	// SSR
	SSR.SubsystemName	:= mpSSQ^.Position;
	SSR.eReturnCode	:= E_ErrorConv.SubsystemNUMBER_UNKNOWN;

	// Reject telegram	
	M_SendData(
		meChannel := meChannelSrc,
		mMsgType  := E_ITC_MsgTypeConv.SUBSYSTEM_STATUS_REPORT,
		mpData    := ADR(SSR),
		mLen	  := SIZEOF(SSR));
		
	// Unknown SubSystem number received
	DebugMsg := CONCAT('SSQ, unknown SubSystem name received: ', mpSSQ^.Position);
	fbDebugMsg.M_SendErrorMsg(mMessage := DebugMsg);
END_IF
END_METHOD

METHOD PROTECTED M_ProcessTDQ : BOOL
(**************************************************************************************
 *  Application     :   BoxControl Framework
 *  Revision date   :   $Date: 2021-04-08 12:45:11 +0200 (tor, 08 apr 2021) $
 *  Author          :   CDC
 * ------------------------------------------------------------------------------------
 *  © Swisslog AG
 *  Swisslog is not liable for any usage of this source code that is not agreed 
 *  on between Swisslog and the other party. The mandatory legal liability remains 
 *  unaffected.
 * ------------------------------------------------------------------------------------
 *  Revision History: 
 *
 *  VERSION DATE         INITIALS     DESCRIPTION
 *  0.0     DD.MM.YYYY   (name)       (explain customized modifications)
 *
 **************************************************************************************)
VAR_INPUT
	meChannelSrc			: E_MFCS_Channel; // Source communicaton channel
	mpTDQ					: POINTER TO ST_ITC_TDQ; // Pointer to TDQ
	mLen					: UDINT; // Data length
END_VAR

VAR
	mPosition				: ST_PositionIdent ; // Position
	mReturnCode				: E_ErrorConv; // Return code
	mTU_ID_Present			: BOOL; // TU-ID present
	mTU_DataIndex			: DINT; // TU-data index
	mAssignmentID_Present	: BOOL; // Assignment-ID present
	mAssignmentID_Index		: DINT; // Assignment-ID index
END_VAR
// Init
mReturnCode := E_ErrorConv.NO_ERROR_CODE;
M_ProcessTDQ := TRUE;
mTU_ID_Present := FALSE;
mTU_DataIndex := 0;
mAssignmentID_Present := FALSE;
mAssignmentID_Index := 0;

// Get position from telegram
mPosition := F_SearchFunctionPosition( Position := mpTDQ^.Position);

// Order to delete all TU-data
IF mpTDQ^.Code = 1 THEN
	// Check no function number and unknown TU-ID
	IF mpTDQ^.TU_ID = Conveyor.TU_ID_UNKNOWN AND mPosition.eFunctionNumber = 0 THEN
		// Check all TU-Data for DataSets
		FOR mTU_DataIndex := 1 TO Conveyor.NUMBER_OF_TU_DATA BY 1 DO
			// Check if TU-DataSet is used
			IF TU_DataTable[mTU_DataIndex].DataSet.DataPresent THEN	
				// debug message: '11-001-0095-01-1,  TU_DataIndex deleted,  telegram = TDQ,  TU_DataIndex = 5,  TuID = 000012345,  AssignmentID = 999999999'
				DebugMsg := '';
				DebugMsg := CONCAT(DebugMsg, F_AddDividerToSisString(mpTDQ^.Position));
				DebugMsg := CONCAT(DebugMsg, ',  TU_DataIndex deleted');
				DebugMsg := CONCAT(DebugMsg, DebugTextBlocks.TELEGRAM);
				DebugMsg := CONCAT(DebugMsg, 'TDQ');
				DebugMsg := CONCAT(DebugMsg, F_CreateTU_DataString(TU_DataIndex:= mTU_DataIndex));
				fbDebugMsg.M_SendInfoMsg(DebugMsg);
				// Delete TU-Data
				F_DeleteTU_Data(
					TU_DataIndex 	:= mTU_DataIndex, // TU_DataIndex from zone
					NoTTC 			:= FALSE); // No TTC will be sent
			END_IF
		END_FOR

		TDR.Position := mpTDQ^.Position;
		TDR.TU_ID := mpTDQ^.TU_ID;
		TDR.AssignmentID := mpTDQ^.AssignmentID;
		TDR.MsgSequence := mpTDQ^.MsgSequence;
		TDR.ReturnCode := mReturnCode;
		
		M_SendData(
			meChannel := meChannelSrc, 
			mMsgType  := E_ITC_MsgTypeConv.TASK_DELETE_REPORT, 
			mpData    := ADR(TDR),
			mLen	  := SIZEOF(TDR));
		RETURN;
	ELSE
		// Error: Wrong value
		mReturnCode := E_ErrorConv.WRONG_VALUE;
	END_IF
	
// Specific request for TU-ID or position
ELSE
	// Check if an Assignment-ID is present
	mAssignmentID_Present := mpTDQ^.AssignmentID > 0 AND mpTDQ^.AssignmentID < Conveyor.ASSIGNMENT_ID_UNKNOWN;
	
	// Check if a TU-ID is present
	mTU_ID_Present := mpTDQ^.TU_ID <> F_StuffString('', Conveyor.TU_ID_STRINGLENGTH,'0', FALSE) AND
				      mpTDQ^.TU_ID <> F_StuffString('', Conveyor.TU_ID_STRINGLENGTH,' ', FALSE);
	
	// If a valid position is found
	IF mPosition.eFunctionNumber > E_FunctionNumber.F_BEGIN_FUNCTION AND
	   mPosition.ZoneNumber > 0 THEN
		// Get TU-data from zone
		mTU_DataIndex := F_GetTU_DataIndex(
								eFunctionNumber := mPosition.eFunctionNumber, // PositionNumber
								ZoneNumber := mPosition.ZoneNumber); // ZoneNumber
		// A TU index was found
		IF mTU_DataIndex > 0 THEN
			IF mAssignmentID_Present THEN
				// Compare received Assignment ID with the Assignment ID from the position
				IF TU_DataTable[mTU_DataIndex].AssignmentID <> mpTDQ^.AssignmentID THEN
					// Error: Wrong Assignement-ID
					mReturnCode := E_ErrorConv.ASSIGNMENT_ID_WRONG;
				END_IF
			ELSIF mTU_ID_Present THEN
				// Compare received TU ID with the TU ID from the position
				IF TU_DataTable[mTU_DataIndex].TU_ID.ASCII <> mpTDQ^.TU_ID THEN
					// Error: Wrong TU-ID
					mReturnCode := E_ErrorConv.TU_ID_WRONG;
				END_IF
			ELSE
				// Error: Wrong value
				mReturnCode := E_ErrorConv.ID_WRONG;
			END_IF
		ELSE
			// Error: No TU data set available on position
			mReturnCode := E_ErrorConv.EMPTY_TU_DATA_SET;
		END_IF
		
	// Request to subsystem
	ELSIF mpTDQ^.Position <> F_ReduceToAlphaNumeric(SubsystemRegistry.SubsystemName) THEN
		// Error: Position wrong 
		mReturnCode := E_ErrorConv.FUNCTIONNUMBER_UNKNOWN;
		
	// Telegram without function number
	ELSE
		IF mAssignmentID_Present THEN
			// Search TU-data index based on the Assignement-ID in the TU-data table
			mAssignmentID_Index := F_SearchAssignmentId(mpTDQ^.AssignmentID);
		END_IF
		
		IF mTU_ID_Present THEN
			// Search TU-data index based on the TU-ID in the TU-data table
			mTU_DataIndex := F_SearchTU_ByHashCode(mpTDQ^.TU_ID);
		END_IF			
		
		// If an Assignement-ID index is found
		IF mAssignmentID_Index <> 0 THEN
			// Search position belonging to the Assignement-ID index
			// to report last position
			mPosition := F_SearchPositionOfTU_Index(
								TU_DataIndex := mAssignmentID_Index, // TU_DataIndex from zone
								eStartFunctionNumber := E_FunctionNumber.F_BEGIN_FUNCTION + 1); // Start Zone
		// If a TU-data index is found
		ELSIF mTU_DataIndex <> 0 THEN
			// Search position belonging to the TU-data index
			// to report last position
			mPosition := F_SearchPositionOfTU_Index(
								TU_DataIndex := mTU_DataIndex, // TU_DataIndex from zone
								eStartFunctionNumber := E_FunctionNumber.F_BEGIN_FUNCTION + 1); // Start Zone
		ELSE
			IF mAssignmentID_Present THEN
				// Error: Wrong Assignement-ID
				mReturnCode := E_ErrorConv.ASSIGNMENT_ID_WRONG;
			ELSIF mTU_ID_Present THEN
				// Error: Wrong TU-ID
				mReturnCode := E_ErrorConv.TU_ID_WRONG;
			ELSE
				// Error: No data
				mReturnCode := E_ErrorConv.ID_WRONG;
			END_IF
		END_IF
	END_IF
END_IF

// Send task delete report
IF mPosition.eFunctionNumber <> E_FunctionNumber.F_BEGIN_FUNCTION THEN
	TDR.Position := F_ReduceToAlphaNumeric(FunctionRegistry[mPosition.eFunctionNumber].Zone[mPosition.ZoneNumber].ZoneName);
ELSE
	TDR.Position := mpTDQ^.Position;
END_IF
TDR.TU_ID := mpTDQ^.TU_ID;
TDR.AssignmentID := mpTDQ^.AssignmentID;
TDR.MsgSequence := mpTDQ^.MsgSequence;
TDR.ReturnCode := mReturnCode;

M_SendData(
	meChannel := meChannelSrc, 
	mMsgType  := E_ITC_MsgTypeConv.TASK_DELETE_REPORT, 
	mpData    := ADR(TDR),
	mLen	  := SIZEOF(TDR));

// Still no error so far
IF mReturnCode = 0  THEN
	// TU-data index available
	IF mTU_DataIndex <> 0 THEN
		// debug message: '11-001-0095-01-1,  TU_DataIndex deleted,  telegram = TDQ,  TU_DataIndex = 5,  TuID = 000012345,  AssignmentID = 999999999'
		DebugMsg := '';
		DebugMsg := CONCAT(DebugMsg, F_AddDividerToSisString(mpTDQ^.Position));
		DebugMsg := CONCAT(DebugMsg, ',  TU_DataIndex deleted');
		DebugMsg := CONCAT(DebugMsg, DebugTextBlocks.TELEGRAM);
		DebugMsg := CONCAT(DebugMsg, 'TDQ');
		DebugMsg := CONCAT(DebugMsg, F_CreateTU_DataString(TU_DataIndex:= mTU_DataIndex));
		fbDebugMsg.M_SendInfoMsg(DebugMsg);
		// Delete TU-data in the system
		F_DeleteTU_Data(
			TU_DataIndex 	:= mTU_DataIndex,
			NoTTC 			:= FALSE);
	// Assignement-ID index available
	ELSIF mAssignmentID_Index <> 0 THEN
		// debug message: '11-001-0095-01-1,  TU_DataIndex deleted,  telegram = TDQ,  TU_DataIndex = 5,  TuID = 000012345,  AssignmentID = 999999999'
		DebugMsg := '';
		DebugMsg := CONCAT(DebugMsg, F_AddDividerToSisString(mpTDQ^.Position));
		DebugMsg := CONCAT(DebugMsg, ',  TU_DataIndex deleted');
		DebugMsg := CONCAT(DebugMsg, DebugTextBlocks.TELEGRAM);
		DebugMsg := CONCAT(DebugMsg, 'TDQ');
		DebugMsg := CONCAT(DebugMsg, F_CreateTU_DataString(TU_DataIndex:= mAssignmentID_Index));
		fbDebugMsg.M_SendInfoMsg(DebugMsg);
		// Delete TU-data in the system
		F_DeleteTU_Data(
			TU_DataIndex 	:= mAssignmentID_Index,
			NoTTC 			:= FALSE);
	ELSE		
		DebugMsg := 'TDQ, Process failed - no TU-index available.';
		fbDebugMsg.M_SendErrorMsg(mMessage := DebugMsg);		
	END_IF
END_IF
END_METHOD

METHOD PROTECTED M_ProcessToElement : BOOL
(**************************************************************************************
 * 	Application		:	BoxControl Framework
 *	Revision		:	$Revision: 474929 $
 *	Revision date	:	$Date: 2021-04-08 12:45:11 +0200 (tor, 08 apr 2021) $
 *	Last changed by	:	$Author: b7gessa $
 *	URL				:	$URL: http://almscdc.swisslog.com/repo/SWPD/Development/BoxControlFramework/20_Release/tags/R1.12.0/01_Software/BCF/BCF/JumpStart/20_Product/10_BCF/11_Conv/11_Com/11_ITC/FB_ITC_Conveyor.TcPOU $
 *
 *	Purpose			:	ITC - Process message to element
 *
 * ------------------------------------------------------------------------------------
 *	Copyright Swisslog [IP AG], Switzerland. All rights reserved.
 * 
 * ------------------------------------------------------------------------------------
 *	
 * 	Revision History: 
 *
 * 	VERSION			DATE			INITIALS			DESCRIPTION
 *	0.1				01.01.2001		swl					Example
 *
 **************************************************************************************)
VAR_INPUT
	meElementNumber	: E_ElementNumber;
	meChannelSrc	: E_MFCS_Channel; // Source communicaton channel
	mMsgType			: INT; // msg type
	mpData				: POINTER TO PVOID; // data pointer
	mLen				: UDINT; // Data length
END_VAR

VAR
	mrefObject		: REFERENCE TO FB_BaseObject; // Reference
END_VAR
// Initialize
M_ProcessToElement := TRUE;

// Check if ElementNumber is valid
IF meElementNumber > E_ElementNumber.E_BEGIN_ELEMENT AND 
   meElementNumber < E_ElementNumber.E_END_ELEMENT THEN
	// Set reference
	mrefObject REF= ElementRegistry[meElementNumber].rElement;
	
	// Check if reference is valid
	IF __ISVALIDREF(mrefObject) THEN
			// Forward message to corresponding object
		M_ProcessToElement := mrefObject.M_ITC_ProcessMsg(
								meChannelSrc := meChannelSrc,
								mMsgType	 := mMsgType,
								mpData		 := mpData,
								mLen		 := mLen); 
	END_IF	
END_IF
END_METHOD

METHOD PROTECTED M_ProcessToFunction : BOOL
(**************************************************************************************
 * 	Application		:	BoxControl Framework
 *	Revision		:	$Revision: 474929 $
 *	Revision date	:	$Date: 2021-04-08 12:45:11 +0200 (tor, 08 apr 2021) $
 *	Last changed by	:	$Author: b7gessa $
 *	URL				:	$URL: http://almscdc.swisslog.com/repo/SWPD/Development/BoxControlFramework/20_Release/tags/R1.12.0/01_Software/BCF/BCF/JumpStart/20_Product/10_BCF/11_Conv/11_Com/11_ITC/FB_ITC_Conveyor.TcPOU $
 *
 *	Purpose			:	ITC - Process message to function
 *
 * ------------------------------------------------------------------------------------
 *	Copyright Swisslog [IP AG], Switzerland. All rights reserved.
 * 
 * ------------------------------------------------------------------------------------
 *	
 * 	Revision History: 
 *
 * 	VERSION			DATE			INITIALS			DESCRIPTION
 *	0.1				01.01.2001		swl					Example
 *
 **************************************************************************************)
VAR_INPUT
	meFunctionNumber	: E_FunctionNumber; // Function number
	meChannelSrc		: E_MFCS_Channel; // Source communicaton channel
	mMsgType			: INT; // msg type
	mpData				: POINTER TO PVOID; // data pointer
	mLen				: UDINT; // Data length
END_VAR

VAR
	mrefObject			: REFERENCE TO FB_BaseObject; // Reference
END_VAR
// Initialize
M_ProcessToFunction := TRUE;

// If a valid function was found with a valid zone
IF 	meFunctionNumber > E_FunctionNumber.F_BEGIN_FUNCTION AND 
	meFunctionNumber < E_FunctionNumber.F_END_FUNCTION THEN

	// Set reference 
	mrefObject REF= FunctionRegistry[meFunctionNumber].rFunction;
	
	// Check if reference is valid
	IF __ISVALIDREF(mrefObject) THEN

		// Call M_ITC_AddToBuffer
		M_ProcessToFunction := mrefObject.M_ITC_ProcessMsg(
								meChannelSrc := meChannelSrc, // Number of the source 
								mMsgType	 := mMsgType, // Type of the ITC message
								mpData		 := mpData,
								mLen		 := mLen); // Data pointer of the message	
	END_IF
END_IF
END_METHOD

METHOD PROTECTED M_ProcessToGroup : BOOL
(**************************************************************************************
 * 	Application		:	BoxControl Framework
 *	Revision		:	$Revision: 474929 $
 *	Revision date	:	$Date: 2021-04-08 12:45:11 +0200 (tor, 08 apr 2021) $
 *	Last changed by	:	$Author: b7gessa $
 *	URL				:	$URL: http://almscdc.swisslog.com/repo/SWPD/Development/BoxControlFramework/20_Release/tags/R1.12.0/01_Software/BCF/BCF/JumpStart/20_Product/10_BCF/11_Conv/11_Com/11_ITC/FB_ITC_Conveyor.TcPOU $
 *
 *	Purpose			:	ITC - Process message to group
 *
 * ------------------------------------------------------------------------------------
 *	Copyright Swisslog [IP AG], Switzerland. All rights reserved.
 * 
 * ------------------------------------------------------------------------------------
 *	
 * 	Revision History: 
 *
 * 	VERSION			DATE			INITIALS			DESCRIPTION
 *	0.1				01.01.2001		swl					Example
 *
 **************************************************************************************)
VAR_INPUT
	meGroupNumber		: E_GroupNumber; // Groupnumber
	meChannelSrc		: E_MFCS_Channel; // Source communicaton channel
	mMsgType			: INT; // msg type
	mpData				: POINTER TO PVOID; // data pointer
	mLen				: UDINT; // Data length
END_VAR

VAR
	mrefObject			: REFERENCE TO FB_BaseObject; // Reference
END_VAR
// Initialize
M_ProcessToGroup := TRUE;

// Check if GroupNumber is valid
IF meGroupNumber > E_GroupNumber.G_BEGIN_GROUP AND 
   meGroupNumber < E_GroupNumber.G_END_GROUP THEN
	// Set reference
	mrefObject REF= GroupRegistry[meGroupNumber].rGroup;
	
	// Check if reference is valid
	IF __ISVALIDREF(mrefObject) THEN
		
		// Send ITC-message to a specified group
		M_ProcessToGroup := mrefObject.M_ITC_ProcessMsg(
								meChannelSrc := meChannelSrc,
								mMsgType	 := mMsgType, 
								mpData		 := mpData,
								mLen		 := mLen); 
	END_IF
END_IF
END_METHOD

METHOD PROTECTED M_ProcessToSubsystem : BOOL
(**************************************************************************************
 * 	Application		:	BoxControl Framework
 *	Revision		:	$Revision: 474929 $
 *	Revision date	:	$Date: 2021-04-08 12:45:11 +0200 (tor, 08 apr 2021) $
 *	Last changed by	:	$Author: b7gessa $
 *	URL				:	$URL: http://almscdc.swisslog.com/repo/SWPD/Development/BoxControlFramework/20_Release/tags/R1.12.0/01_Software/BCF/BCF/JumpStart/20_Product/10_BCF/11_Conv/11_Com/11_ITC/FB_ITC_Conveyor.TcPOU $
 *
 *	Purpose			:	ITC - Process message to subsystem
 *
 * ------------------------------------------------------------------------------------
 *	Copyright Swisslog [IP AG], Switzerland. All rights reserved.
 * 
 * ------------------------------------------------------------------------------------
 *	
 * 	Revision History: 
 *
 * 	VERSION			DATE			INITIALS			DESCRIPTION
 *	0.1				01.01.2001		swl					Example
 *
 **************************************************************************************)
VAR_INPUT
	meChannelSrc		: E_MFCS_Channel; // Source communicaton channel
	mMsgType			: INT; // msg type
	mpData				: POINTER TO PVOID; // data pointer
	mLen				: UDINT; // Data length
END_VAR

VAR
	mrefObject			: REFERENCE TO FB_BaseObject; // Reference
END_VAR
// Initialize
M_ProcessToSubsystem := TRUE;

// Set reference 
mrefObject REF= SubsystemRegistry.rSubsystem;

// Check if reference is valid
IF __ISVALIDREF(mrefObject) THEN
	// Call M_ITC_AddToBuffer
	M_ProcessToSubsystem := mrefObject.M_ITC_ProcessMsg(
								meChannelSrc := meChannelSrc,
								mMsgType	 := mMsgType, 
								mpData		 := mpData,	
								mLen		 := mLen);  
END_IF
END_METHOD

METHOD PROTECTED M_ProcessTTA : BOOL
(**************************************************************************************
 * 	Application		:	BoxControl Framework
 *	Revision		:	$Revision: 474929 $
 *	Revision date	:	$Date: 2021-04-08 12:45:11 +0200 (tor, 08 apr 2021) $
 *	Last changed by	:	$Author: b7gessa $
 *	URL				:	$URL: http://almscdc.swisslog.com/repo/SWPD/Development/BoxControlFramework/20_Release/tags/R1.12.0/01_Software/BCF/BCF/JumpStart/20_Product/10_BCF/11_Conv/11_Com/11_ITC/FB_ITC_Conveyor.TcPOU $
 *
 *	Purpose			:	Process a received Transport Task Assignment telegram.
 *
 * ------------------------------------------------------------------------------------
 *	Copyright Swisslog [IP AG], Switzerland. All rights reserved.
 * 
 * ------------------------------------------------------------------------------------
 *	
 * 	Revision History: 
 *
 * VERSION DATE         INITIALS     DESCRIPTION
 * 0.0     DD.MM.YYYY   (name)       (explain customized modifications)
 *
 **************************************************************************************)
VAR_INPUT
	meChannelSrc				: E_MFCS_Channel; // Source communicaton channel
	mpTTA						: POINTER TO ST_ITC_TTA; // Pointer to TTA
	mLen						: UDINT;
END_VAR

VAR
	mOtherPosition				: ST_PositionIdent; // OtherPosition where same Index is used
	mDestinationPosition		: ARRAY[1..NUMBER_OF_DESTINATIONS] OF ST_PositionIdent; // DestinationPosition
	mVirtualDestinationPosition	: ARRAY[1..NUMBER_OF_DESTINATIONS] OF ST_PositionIdent;
	mReturnCode					: E_ErrorConv; // Error code
	mTU_DataIndexPosition		: DINT; // Data Index from PositionNumber
	mTU_DataIndex				: DINT; // Data Index from Data_ID
	mRequestForPosition			: BOOL; // Request for a Position
	mTransportData				: ST_TransportControlData; // Transport data
	mTU_ID_Present				: BOOL; // TU-ID present
	mAssignmentID_Present		: BOOL; // Assignment ID present
	mAssignmentID_Index			: DINT; // Assignment ID index
	mDestIndex					: INT; // Temporary destination index
END_VAR
// Initialize
M_ProcessTTA := TRUE;
mTU_DataIndexPosition := 0;
mRequestForPosition := FALSE;	
mTU_DataIndex := 0;
mAssignmentID_Index := 0;
mAssignmentID_Present := FALSE;
mTU_ID_Present := FALSE;

(**************************************************************************************
Check if request is valid
***************************************************************************************)
// Search position in registry
Position := F_SearchFunctionPosition(Position := mpTTA^.Position);

//Check if a TU-ID is present
mTU_ID_Present := 	mpTTA^.TU_ID <> F_StuffString('', Conveyor.TU_ID_STRINGLENGTH,'0', FALSE)
				AND mpTTA^.TU_ID <> F_StuffString('', Conveyor.TU_ID_STRINGLENGTH,' ', FALSE);

IF mTU_ID_Present THEN
	// Search if the TU-ID already exists
	mTU_DataIndex := F_SearchTU_ByHashCode(mpTTA^.TU_ID);
END_IF	

// Check if an asssignment-ID is present					   
mAssignmentID_Present := mpTTA^.AssignmentID > 0;

IF mAssignmentID_Present THEN
	// Search if the assignment-ID already exists
	mAssignmentID_Index := F_SearchAssignmentId(mpTTA^.AssignmentID);
END_IF


// If the telegram contains no TU-ID and no assignment-ID
IF NOT mTU_ID_Present AND NOT mAssignmentID_Present THEN
	// Error: ID is wrong 
	mReturnCode := E_ErrorConv.ID_WRONG;
	// debug message: '11-000-0000-00-0,  TuID and AssignmentID missing,  telegram = TTA'
	DebugMsg:= '';
	DebugMsg:= CONCAT(DebugMsg, F_AddDividerToSisString(SubsystemRegistry.SubsystemName));
	DebugMsg:= CONCAT(DebugMsg, ',  TuID and AssignmentID missing');
	DebugMsg:= CONCAT(DebugMsg, DebugTextBlocks.TELEGRAM);
	DebugMsg:= CONCAT(DebugMsg, 'TTA');
	fbDebugMsg.M_SendErrorMsg(mMessage := DebugMsg);


// If the request goes to a position
ELSIF Position.eFunctionNumber > E_FunctionNumber.F_BEGIN_FUNCTION AND 
	Position.eFunctionNumber < E_FunctionNumber.F_END_FUNCTION THEN
	// If a valid zone was found
	IF 	Position.ZoneNumber > 0
	AND Position.ZoneNumber <= NUMBER_OF_ZONES_PER_FUNCTION THEN
		// Get transport data
		mTransportData := F_GetTransportControlData(
		eFunctionNumber := Position.eFunctionNumber,
		ZoneNumber		:= Position.ZoneNumber);
		
		(*	Data can only be added if the location is physically occupied.
			State occupied is not working in this place, because on a system
			with enabled MFC, the place gets occupied only with a physical 
			and a logical unit. *)
		IF mTransportData.SensorOccupied THEN
			// Save - Valid request for a position
			mRequestForPosition := TRUE;	

			// Get TU Index of telegram position
			mTU_DataIndexPosition := F_GetTU_DataIndex( 
			eFunctionNumber := Position.eFunctionNumber,
			ZoneNumber 		:= Position.ZoneNumber);
			// If an index is found
			IF mTU_DataIndexPosition > 0 THEN
			(* 
			Adding data is allowed, if
			- TU-ID of desired position is 'unknown' OR
			- Telegram TU-ID is equal to position TU-ID
			
			AND
			- Position consists of an unknown assignment-ID OR
			- Assignment-ID is equal to the requested one		
			
			AND
			- When a requested Index was available, it needs to be equal to position index		
			*)
				IF (TU_DataTable[mTU_DataIndexPosition].TU_ID.ASCII = Conveyor.TU_ID_UNKNOWN OR 
				mpTTA^.TU_ID = TU_DataTable[mTU_DataIndexPosition].TU_ID.ASCII) AND 
				(mpTTA^.AssignmentID = TU_DataTable[mTU_DataIndexPosition].AssignmentID OR
				Conveyor.ASSIGNMENT_ID_UNKNOWN = TU_DataTable[mTU_DataIndexPosition].AssignmentID) AND
				((mpTTA^.TU_DataIndex > 0 AND mpTTA^.TU_DataIndex = mTU_DataIndexPosition) OR (mpTTA^.TU_DataIndex = 0)) THEN 
					// Adding data is allowed by TU-ID
					;
				// Adding not allowed
				ELSE
					// When the assignment-ID was not equal to the already existing or 
					// the assignment-ID on the position was not unknown
					IF TU_DataTable[mTU_DataIndexPosition].AssignmentID <> mpTTA^.AssignmentID AND 
					   TU_DataTable[mTU_DataIndexPosition].AssignmentID <> Conveyor.ASSIGNMENT_ID_UNKNOWN THEN
						// Error: Assignment-ID is false 
						mReturnCode := E_ErrorConv.ASSIGNMENT_ID_WRONG;
						// debug message: '11-001-0120-01-0,  AssignmentID mismatch,  telegram = TTA,  expected = 112233,  current = 332211'
						DebugMsg:= '';
						DebugMsg:= CONCAT(DebugMsg, F_AddDividerToSisString(Position.PositionName));
						DebugMsg:= CONCAT(DebugMsg, ',  AssignmentID mismatch');
						DebugMsg:= CONCAT(DebugMsg, DebugTextBlocks.TELEGRAM);
						DebugMsg:= CONCAT(DebugMsg, 'TTA');
						DebugMsg:= CONCAT(DebugMsg, DebugTextBlocks.EXPECTED);
						DebugMsg:= CONCAT(DebugMsg, UDINT_TO_STRING(TU_DataTable[mTU_DataIndexPosition].AssignmentID) );
						DebugMsg:= CONCAT(DebugMsg, DebugTextBlocks.CURRENT);
						DebugMsg:= CONCAT(DebugMsg, UDINT_TO_STRING(mpTTA^.AssignmentID) );
						fbDebugMsg.M_SendErrorMsg(mMessage := DebugMsg);

					// Otherwise its because of a wrong TU-ID
					// - Not equal
					// - Not unknown
					ELSIF TU_DataTable[mTU_DataIndexPosition].TU_ID.ASCII <> Conveyor.TU_ID_UNKNOWN AND 
						  TU_DataTable[mTU_DataIndexPosition].TU_ID.ASCII <> mpTTA^.TU_ID THEN
						// Error: TU-ID is false 
						mReturnCode := E_ErrorConv.TU_ID_WRONG;
						// debug message: '11-001-0120-01-0,  TuID mismatch,  telegram = TTA,  expected = 112233,  current = 332211'
						DebugMsg:= '';
						DebugMsg:= CONCAT(DebugMsg, F_AddDividerToSisString(Position.PositionName));
						DebugMsg:= CONCAT(DebugMsg, ',  TuID mismatch');
						DebugMsg:= CONCAT(DebugMsg, DebugTextBlocks.TELEGRAM);
						DebugMsg:= CONCAT(DebugMsg, 'TTA');
						DebugMsg:= CONCAT(DebugMsg, DebugTextBlocks.EXPECTED);
						DebugMsg:= CONCAT(DebugMsg, TU_DataTable[mTU_DataIndexPosition].TU_ID.ASCII);
						DebugMsg:= CONCAT(DebugMsg, DebugTextBlocks.CURRENT);
						DebugMsg:= CONCAT(DebugMsg, mpTTA^.TU_ID);
						fbDebugMsg.M_SendErrorMsg(mMessage := DebugMsg);

					// Otherwise, requested index was wrong
					ELSE
						mReturnCode := E_ErrorConv.WRONG_VALUE;
						// debug message: '11-001-0120-01-0,  TU_DataIndex mismatch,  telegram = TTA,  expected = 1,  current = 3'
						DebugMsg:= '';
						DebugMsg:= CONCAT(DebugMsg, F_AddDividerToSisString(Position.PositionName));
						DebugMsg:= CONCAT(DebugMsg, ',  TU_DataIndex mismatch');
						DebugMsg:= CONCAT(DebugMsg, DebugTextBlocks.TELEGRAM);
						DebugMsg:= CONCAT(DebugMsg, 'TTA');
						DebugMsg:= CONCAT(DebugMsg, DebugTextBlocks.EXPECTED);
						DebugMsg:= CONCAT(DebugMsg, DINT_TO_STRING(mTU_DataIndexPosition)  );
						DebugMsg:= CONCAT(DebugMsg, DebugTextBlocks.CURRENT);
						DebugMsg:= CONCAT(DebugMsg, DINT_TO_STRING(mpTTA^.TU_DataIndex)  );
						fbDebugMsg.M_SendErrorMsg(mMessage := DebugMsg);
					END_IF		
				END_IF
			END_IF 
		ELSE
			// Error: Zone free
			mReturnCode := E_ErrorConv.POSITION_NOT_CORRECT_OCCUPIED;
			// debug message: '11-001-0120-01-0,  position is not occupied,  telegram = TTA'
			DebugMsg:= '';
			DebugMsg:= CONCAT(DebugMsg, F_AddDividerToSisString(Position.PositionName));
			DebugMsg:= CONCAT(DebugMsg, ',  position is not occupied');
			DebugMsg:= CONCAT(DebugMsg, DebugTextBlocks.TELEGRAM);
			DebugMsg:= CONCAT(DebugMsg, 'TTA');
			fbDebugMsg.M_SendErrorMsg(mMessage := DebugMsg);
		END_IF

	ELSE
		// Error: Position wrong 
		mReturnCode := E_ErrorConv.FUNCTIONNUMBER_UNKNOWN;
		// debug message: '11-000-0000-00-0,  unknown position addressed,  telegram = TTA,  Position = 99-999-9999-99-9'
		DebugMsg:= '';
		DebugMsg:= CONCAT(DebugMsg, F_AddDividerToSisString(SubsystemRegistry.SubsystemName));
		DebugMsg:= CONCAT(DebugMsg, ',  unknown position addressed');
		DebugMsg:= CONCAT(DebugMsg, DebugTextBlocks.TELEGRAM);
		DebugMsg:= CONCAT(DebugMsg, 'TTA');
		DebugMsg:= CONCAT(DebugMsg, DebugTextBlocks.POSITION);
		DebugMsg:= CONCAT(DebugMsg, F_AddDividerToSisString(Name:= mpTTA^.Position)  );
		fbDebugMsg.M_SendErrorMsg(mMessage := DebugMsg);
	END_IF

// If the request goes to the subsystem MM-000-0000-00-0
ELSIF NOT F_EqualSisNames(Name1:= mpTTA^.Position,
						  Name2:= SubsystemRegistry.SubsystemName) THEN
	// Error: Position wrong 
	mReturnCode := E_ErrorConv.FUNCTIONNUMBER_UNKNOWN; 
	// debug message: '00-000-0000-00-0,  unknown position addressed,  telegram = TTA,  Position = 99-999-9999-99-9'
	DebugMsg:= '';
	DebugMsg:= CONCAT(DebugMsg, '00-000-0000-00-0');  // subsystem is not properly addressed
	DebugMsg:= CONCAT(DebugMsg, ',  unknown position addressed');
	DebugMsg:= CONCAT(DebugMsg, DebugTextBlocks.TELEGRAM);
	DebugMsg:= CONCAT(DebugMsg, 'TTA');
	DebugMsg:= CONCAT(DebugMsg, DebugTextBlocks.POSITION);
	DebugMsg:= CONCAT(DebugMsg, F_AddDividerToSisString(Name:= mpTTA^.Position)  );
	fbDebugMsg.M_SendErrorMsg(mMessage := DebugMsg);

// TU-data index update request to subsystem
ELSIF mpTTA^.TU_DataIndex > 0 THEN
	// Validate corresponding index
	IF TU_DataTable[mpTTA^.TU_DataIndex].DataSet.DataPresent THEN
		(* If the received telegram contains two existing IDs (Assignment and TU) -> both have to match to the same index. *)
		IF mTU_DataIndex > 0 AND mAssignmentID_Index > 0 THEN
			IF mTU_DataIndex <> mAssignmentID_Index THEN
				mReturnCode := E_ErrorConv.WRONG_VALUE;	
				// debug message: '11-000-0000-00-0,  AssignmentID mismatch,  telegram = TTA,  expected = 87654321,  current = 12345678'
				DebugMsg:= '';
				DebugMsg:= CONCAT(DebugMsg, F_AddDividerToSisString(SubsystemRegistry.SubsystemName));
				DebugMsg:= CONCAT(DebugMsg, ',  AssignmentID mismatch');
				DebugMsg:= CONCAT(DebugMsg, DebugTextBlocks.TELEGRAM);
				DebugMsg:= CONCAT(DebugMsg, 'TTA');
				DebugMsg:= CONCAT(DebugMsg, DebugTextBlocks.EXPECTED);
				DebugMsg:= CONCAT(DebugMsg, UDINT_TO_STRING(TU_DataTable[mTU_DataIndex].AssignmentID)  );
				DebugMsg:= CONCAT(DebugMsg, DebugTextBlocks.CURRENT);
				DebugMsg:= CONCAT(DebugMsg, UDINT_TO_STRING(mpTTA^.AssignmentID)  );
				fbDebugMsg.M_SendErrorMsg(mMessage := DebugMsg);

			// Compare found index to TTA index
			ELSIF mpTTA^.TU_DataIndex <> mTU_DataIndex THEN
				mReturnCode := E_ErrorConv.WRONG_VALUE;	
				// debug message: '11-000-0000-00-0,  TU_DataIndex mismatch,  telegram = TTA,  expected = 1,  current = 3'
				DebugMsg:= '';
				DebugMsg:= CONCAT(DebugMsg, F_AddDividerToSisString(SubsystemRegistry.SubsystemName));
				DebugMsg:= CONCAT(DebugMsg, ',  TU_DataIndex mismatch');
				DebugMsg:= CONCAT(DebugMsg, DebugTextBlocks.TELEGRAM);
				DebugMsg:= CONCAT(DebugMsg, 'TTA');
				DebugMsg:= CONCAT(DebugMsg, DebugTextBlocks.EXPECTED);
				DebugMsg:= CONCAT(DebugMsg, DINT_TO_STRING(mTU_DataIndex)  );
				DebugMsg:= CONCAT(DebugMsg, DebugTextBlocks.CURRENT);
				DebugMsg:= CONCAT(DebugMsg, DINT_TO_STRING(mpTTA^.TU_DataIndex)  );
				fbDebugMsg.M_SendErrorMsg(mMessage := DebugMsg);
			END_IF

		// When an TU-ID index was found
		ELSIF mTU_DataIndex > 0 THEN
			// Compare found index to TTA index
			IF mTU_DataIndex <> mpTTA^.TU_DataIndex THEN
				mReturnCode := E_ErrorConv.WRONG_VALUE;	
				// debug message: '11-000-0000-00-0,  TU_DataIndex mismatch,  telegram = TTA,  expected = 1,  current = 3'
				DebugMsg:= '';
				DebugMsg:= CONCAT(DebugMsg, F_AddDividerToSisString(SubsystemRegistry.SubsystemName));
				DebugMsg:= CONCAT(DebugMsg, ',  TU_DataIndex mismatch');
				DebugMsg:= CONCAT(DebugMsg, DebugTextBlocks.TELEGRAM);
				DebugMsg:= CONCAT(DebugMsg, 'TTA');
				DebugMsg:= CONCAT(DebugMsg, DebugTextBlocks.EXPECTED);
				DebugMsg:= CONCAT(DebugMsg, DINT_TO_STRING(mTU_DataIndex)  );
				DebugMsg:= CONCAT(DebugMsg, DebugTextBlocks.CURRENT);
				DebugMsg:= CONCAT(DebugMsg, DINT_TO_STRING(mpTTA^.TU_DataIndex)  );
				fbDebugMsg.M_SendErrorMsg(mMessage := DebugMsg);
			END_IF

		// When an assignment-ID index was found
		ELSIF mAssignmentID_Index > 0 THEN
			// Compare found index to TTA index
			IF mAssignmentID_Index <> mpTTA^.TU_DataIndex THEN
				mReturnCode := E_ErrorConv.WRONG_VALUE;	
				// debug message: '11-000-0000-00-0,  AssignmentID mismatch,  telegram = TTA,  expected = 87654321,  current = 12345678'
				DebugMsg:= '';
				DebugMsg:= CONCAT(DebugMsg, F_AddDividerToSisString(SubsystemRegistry.SubsystemName));
				DebugMsg:= CONCAT(DebugMsg, ',  AssignmentID mismatch');
				DebugMsg:= CONCAT(DebugMsg, DebugTextBlocks.TELEGRAM);
				DebugMsg:= CONCAT(DebugMsg, 'TTA');
				DebugMsg:= CONCAT(DebugMsg, DebugTextBlocks.EXPECTED);
				DebugMsg:= CONCAT(DebugMsg, UDINT_TO_STRING(TU_DataTable[mAssignmentID_Index].AssignmentID)  );
				DebugMsg:= CONCAT(DebugMsg, DebugTextBlocks.CURRENT);
				DebugMsg:= CONCAT(DebugMsg, UDINT_TO_STRING(mpTTA^.AssignmentID)  );
				fbDebugMsg.M_SendErrorMsg(mMessage := DebugMsg);
			END_IF
		END_IF

		IF mReturnCode = 0 THEN
			// Validate TU-ID
			IF (TU_DataTable[mpTTA^.TU_DataIndex].TU_ID.ASCII <> Conveyor.TU_ID_UNKNOWN AND mpTTA^.TU_ID <> TU_DataTable[mpTTA^.TU_DataIndex].TU_ID.ASCII)
			 OR(TU_DataTable[mpTTA^.TU_DataIndex].AssignmentID <> Conveyor.ASSIGNMENT_ID_UNKNOWN AND mpTTA^.AssignmentID <> TU_DataTable[mpTTA^.TU_DataIndex].AssignmentID) THEN
				IF (TU_DataTable[mpTTA^.TU_DataIndex].TU_ID.ASCII <> Conveyor.TU_ID_UNKNOWN AND
				mpTTA^.TU_ID <> TU_DataTable[mpTTA^.TU_DataIndex].TU_ID.ASCII) THEN
					// Error: TU-ID is false 
					mReturnCode := E_ErrorConv.TU_ID_WRONG;
					// debug message: '11-001-0120-01-0,  TuID mismatch,  telegram = TTA,  expected = 112233,  current = 332211'
					DebugMsg:= '';
					DebugMsg:= CONCAT(DebugMsg, F_AddDividerToSisString(SubsystemRegistry.SubsystemName));
					DebugMsg:= CONCAT(DebugMsg, ',  TuID mismatch');
					DebugMsg:= CONCAT(DebugMsg, DebugTextBlocks.TELEGRAM);
					DebugMsg:= CONCAT(DebugMsg, 'TTA');
					DebugMsg:= CONCAT(DebugMsg, DebugTextBlocks.EXPECTED);
					DebugMsg:= CONCAT(DebugMsg, TU_DataTable[mpTTA^.TU_DataIndex].TU_ID.ASCII);
					DebugMsg:= CONCAT(DebugMsg, DebugTextBlocks.CURRENT);
					DebugMsg:= CONCAT(DebugMsg, mpTTA^.TU_ID);
					fbDebugMsg.M_SendErrorMsg(mMessage := DebugMsg);

				ELSE
					// Error: Assignment-ID is false 
					mReturnCode := E_ErrorConv.ASSIGNMENT_ID_WRONG;
					// debug message: '11-000-0000-00-0,  AssignmentID mismatch,  telegram = TTA,  expected = 87654321,  current = 12345678'
					DebugMsg:= '';
					DebugMsg:= CONCAT(DebugMsg, F_AddDividerToSisString(SubsystemRegistry.SubsystemName));
					DebugMsg:= CONCAT(DebugMsg, ',  AssignmentID mismatch');
					DebugMsg:= CONCAT(DebugMsg, DebugTextBlocks.TELEGRAM);
					DebugMsg:= CONCAT(DebugMsg, 'TTA');
					DebugMsg:= CONCAT(DebugMsg, DebugTextBlocks.EXPECTED);
					DebugMsg:= CONCAT(DebugMsg, UDINT_TO_STRING(TU_DataTable[mpTTA^.TU_DataIndex].AssignmentID)  );
					DebugMsg:= CONCAT(DebugMsg, DebugTextBlocks.CURRENT);
					DebugMsg:= CONCAT(DebugMsg, UDINT_TO_STRING(mpTTA^.AssignmentID)  );
					fbDebugMsg.M_SendErrorMsg(mMessage := DebugMsg);
				END_IF

			// Checks okay, its allowed to takeover data
			ELSE
				mTU_DataIndex := mpTTA^.TU_DataIndex;
			END_IF
		END_IF
	ELSE
		// Error: No corresponding data set found
		mReturnCode := E_ErrorConv.TU_DATA_INDEX_FREE;
		// debug message: '11-000-0000-00-0,  no corresponding dataset ,  telegram = TTA,  TU_DataIndex = 8'
		DebugMsg:= '';
		DebugMsg:= CONCAT(DebugMsg, F_AddDividerToSisString(SubsystemRegistry.SubsystemName));
		DebugMsg:= CONCAT(DebugMsg, ',  no corresponding dataset');
		DebugMsg:= CONCAT(DebugMsg, DebugTextBlocks.TELEGRAM);
		DebugMsg:= CONCAT(DebugMsg, 'TTA');
		DebugMsg:= CONCAT(DebugMsg, DebugTextBlocks.TU_DATA_INDEX);
		DebugMsg:= CONCAT(DebugMsg, DINT_TO_STRING(mpTTA^.TU_DataIndex)  );
		fbDebugMsg.M_SendErrorMsg(mMessage := DebugMsg);
	
	END_IF
END_IF


(**************************************************************************************
already an error -> cancel processing
***************************************************************************************)
IF mReturnCode <> 0 THEN
	TTC.Position    := mpTTA^.Position;
	TTC.TU_DataIndex:= mTU_DataIndex;
	TTC.MsgSequence := mpTTA^.MsgSequence;
	TTC.TU_ID       := mpTTA^.TU_ID;
	TTC.AssignmentID:= mpTTA^.AssignmentID;
	TTC.ReturnCode  := mReturnCode;
	M_SendData(meChannel:= meChannelSrc, 
	mMsgType := E_ITC_MsgTypeConv.TRANSPORT_TASK_COMPLETE, 
	mpData   := ADR(TTC),
	mLen     := SIZEOF(TTC));
	// debug message already sent
	RETURN;
END_IF


(**************************************************************************************
Check destinations
***************************************************************************************)
// Go through all destinations
FOR Idx := 1 TO mpTTA^.NumberOfDestinations DO			
	mDestinationPosition[Idx] := F_SearchFunctionPosition(Position := mpTTA^.Destination[Idx]);		
	// Check destination is invalid
	IF mDestinationPosition[Idx].eFunctionNumber = E_FunctionNumber.F_BEGIN_FUNCTION THEN
		// Destination invalid
		TTC.Position    := mpTTA^.Position;
		TTC.TU_DataIndex:= mTU_DataIndex;
		TTC.MsgSequence := mpTTA^.MsgSequence;
		TTC.TU_ID       := mpTTA^.TU_ID;
		TTC.AssignmentID:= mpTTA^.AssignmentID;
		TTC.ReturnCode  := E_ErrorConv.DESTINATION_INVALID;
		M_SendData(meChannel:= meChannelSrc, 
		mMsgType := E_ITC_MsgTypeConv.TRANSPORT_TASK_COMPLETE, 
		mpData   := ADR(TTC),
		mLen     := SIZEOF(TTC));
		// debug message: '11-000-0000-00-0,  unknown destination addressed,  telegram = TTA,  destination = 99-999-9999-99-9'
		DebugMsg:= '';
		DebugMsg:= CONCAT(DebugMsg, F_AddDividerToSisString(mpTTA^.Position));
		DebugMsg:= CONCAT(DebugMsg, ',  unknown destination addressed');
		DebugMsg:= CONCAT(DebugMsg, DebugTextBlocks.TELEGRAM);
		DebugMsg:= CONCAT(DebugMsg, 'TTA');
		DebugMsg:= CONCAT(DebugMsg, DebugTextBlocks.DESTINATION);
		DebugMsg:= CONCAT(DebugMsg, F_AddDividerToSisString(mpTTA^.Destination[Idx])  );
		fbDebugMsg.M_SendErrorMsg(mMessage := DebugMsg);
		// debug message just sent
		RETURN;
	END_IF
END_FOR


(**************************************************************************************
Determine TU data index
***************************************************************************************)
(* Adding unknown TU data is only allowed if:
- TU-ID is unknown and no assignment-ID is present
- Assignment-ID is unknown and no TU-ID is present
- Assignment-ID and TU-ID is unknown *)
IF (mpTTA^.TU_ID = Conveyor.TU_ID_UNKNOWN AND NOT mAssignmentID_Present) OR
(mpTTA^.AssignmentID = Conveyor.ASSIGNMENT_ID_UNKNOWN AND NOT mTU_ID_Present) OR
(mpTTA^.TU_ID = TU_ID_UNKNOWN AND mpTTA^.AssignmentID = ASSIGNMENT_ID_UNKNOWN) THEN
	// Unknown requests need to be mandatory sent to a position
	IF NOT mRequestForPosition THEN
		//Error: no position request!
		mReturnCode := E_ErrorConv.TU_ID_WRONG;
		// debug message: '11-000-0000-00-0,  no position request,  telegram = TTA'
		DebugMsg:= '';
		DebugMsg:= CONCAT(DebugMsg, F_AddDividerToSisString(SubsystemRegistry.SubsystemName));
		DebugMsg:= CONCAT(DebugMsg, ',  no position request');
		DebugMsg:= CONCAT(DebugMsg, DebugTextBlocks.TELEGRAM);
		DebugMsg:= CONCAT(DebugMsg, 'TTA');
		fbDebugMsg.M_SendErrorMsg(mMessage := DebugMsg);
	
	// If the corresponding position contains no data
	ELSIF mTU_DataIndexPosition = 0 THEN
		// Try insert TU-Data
		mTU_DataIndex := F_InsertTU_Data(
		eFunctionNumber := Position.eFunctionNumber,
		ZoneNumber 		:= Position.ZoneNumber);

		// No free TU Index was found
		IF mTU_DataIndex = 0 THEN
			// Error: No free TU-DataIndex
			mReturnCode := E_ErrorConv.NO_FREE_TU_DATA_SET;
			// debug message: '11-000-0000-00-0,  no free data index,  telegram = TTA,  TuID = 012345,  AssignmentID = 87654321'
			DebugMsg:= '';
			DebugMsg:= CONCAT(DebugMsg, F_AddDividerToSisString(mpTTA^.Position));
			DebugMsg:= CONCAT(DebugMsg, ',  no free data index');
			DebugMsg:= CONCAT(DebugMsg, DebugTextBlocks.TELEGRAM);
			DebugMsg:= CONCAT(DebugMsg, 'TTA');
			DebugMsg:= CONCAT(DebugMsg, DebugTextBlocks.TUID);
			DebugMsg:= CONCAT(DebugMsg, mpTTA^.TU_ID);
			DebugMsg:= CONCAT(DebugMsg, DebugTextBlocks.ASSIGNMENTID);
			DebugMsg:= CONCAT(DebugMsg, UDINT_TO_STRING(mpTTA^.AssignmentID) );
			fbDebugMsg.M_SendErrorMsg(mMessage := DebugMsg);
		END_IF
	// Otherwise
	ELSE
		// Use existing index
		mTU_DataIndex := mTU_DataIndexPosition;
	END_IF

// Otherwise the telegram contains valid IDs
ELSE
	(* If the received telegram contains two valid
	IDs (Assignment and TU) - both have to be equal to the found index. *)
	IF mTU_DataIndex > 0 AND mAssignmentID_Index > 0 THEN
		IF mTU_DataIndex <> mAssignmentID_Index THEN
			mReturnCode := E_ErrorConv.WRONG_VALUE;	
			// debug message: '11-000-0000-00-0,  AssignmentID mismatch,  telegram = TTA,  expected = 87654321,  current = 12345678'
			DebugMsg:= '';
			DebugMsg:= CONCAT(DebugMsg, F_AddDividerToSisString(mpTTA^.Position));
			DebugMsg:= CONCAT(DebugMsg, ',  AssignmentID mismatch');
			DebugMsg:= CONCAT(DebugMsg, DebugTextBlocks.TELEGRAM);
			DebugMsg:= CONCAT(DebugMsg, 'TTA');
			DebugMsg:= CONCAT(DebugMsg, DebugTextBlocks.EXPECTED);
			DebugMsg:= CONCAT(DebugMsg, UDINT_TO_STRING(TU_DataTable[mTU_DataIndex].AssignmentID)  );
			DebugMsg:= CONCAT(DebugMsg, DebugTextBlocks.CURRENT);
			DebugMsg:= CONCAT(DebugMsg, UDINT_TO_STRING(mpTTA^.AssignmentID)  );
			fbDebugMsg.M_SendErrorMsg(mMessage := DebugMsg);
		END_IF

	// If an index based on the assignment-ID was found
	ELSIF mAssignmentID_Index > 0 THEN
		(*  Check if the TU-ID of the found index is unknown.
		Equal to telegram is not needed, because then an index should be found. *)
		IF TU_DataTable[mAssignmentID_Index].TU_ID.ASCII = Conveyor.TU_ID_UNKNOWN THEN
			// Use assignment index
			mTU_DataIndex := mAssignmentID_Index;
		ELSE
			// TU-ID of the found slot does not match
			mReturnCode := E_ErrorConv.TU_ID_WRONG;	
			// debug message: '11-001-0120-01-0,  TuID mismatch,  telegram = TTA,  expected = 112233,  current = 332211'
			DebugMsg:= '';
			DebugMsg:= CONCAT(DebugMsg, F_AddDividerToSisString(mpTTA^.Position));
			DebugMsg:= CONCAT(DebugMsg, ',  TuID mismatch');
			DebugMsg:= CONCAT(DebugMsg, DebugTextBlocks.TELEGRAM);
			DebugMsg:= CONCAT(DebugMsg, 'TTA');
			DebugMsg:= CONCAT(DebugMsg, DebugTextBlocks.EXPECTED);
			DebugMsg:= CONCAT(DebugMsg, TU_DataTable[mAssignmentID_Index].TU_ID.ASCII);
			DebugMsg:= CONCAT(DebugMsg, DebugTextBlocks.CURRENT);
			DebugMsg:= CONCAT(DebugMsg, mpTTA^.TU_ID);
			fbDebugMsg.M_SendErrorMsg(mMessage := DebugMsg);
		END_IF

	// When an index based on the TU-ID was found
	ELSIF mTU_DataIndex > 0 THEN
		(* Check if the Assignment-ID of the found index is unknown.
		Equal to telegram is not needed, because then an index should be found. *)
		IF TU_DataTable[mTU_DataIndex].AssignmentID = Conveyor.ASSIGNMENT_ID_UNKNOWN THEN
			// Keep index (mTU_DataIndex)
			;
		ELSE
			// TU-ID of the found slot does not match
			mReturnCode := E_ErrorConv.ASSIGNMENT_ID_WRONG;	
			// debug message: '11-000-0000-00-0,  AssignmentID mismatch,  telegram = TTA,  expected = 87654321,  current = 12345678'
			DebugMsg:= '';
			DebugMsg:= CONCAT(DebugMsg, F_AddDividerToSisString(mpTTA^.Position));
			DebugMsg:= CONCAT(DebugMsg, ',  AssignmentID mismatch');
			DebugMsg:= CONCAT(DebugMsg, DebugTextBlocks.TELEGRAM);
			DebugMsg:= CONCAT(DebugMsg, 'TTA');
			DebugMsg:= CONCAT(DebugMsg, DebugTextBlocks.EXPECTED);
			DebugMsg:= CONCAT(DebugMsg, UDINT_TO_STRING(TU_DataTable[mTU_DataIndex].AssignmentID)  );
			DebugMsg:= CONCAT(DebugMsg, DebugTextBlocks.CURRENT);
			DebugMsg:= CONCAT(DebugMsg, UDINT_TO_STRING(mpTTA^.AssignmentID)  );
			fbDebugMsg.M_SendErrorMsg(mMessage := DebugMsg);
		END_IF
	END_IF

	IF mReturnCode = 0 THEN
		// If a data index is found
		IF mTU_DataIndex > 0 THEN
			// If the request is for a position
			IF mRequestForPosition THEN
				// Check if this index belongs already to a position	
				mOtherPosition :=	F_SearchPositionOfTU_Index( 
				TU_DataIndex 			:= mTU_DataIndex,
				eStartFunctionNumber	:= E_FunctionNumber.F_BEGIN_FUNCTION);
				
				// If the index was found on another position
				IF (mOtherPosition.eFunctionNumber > E_FunctionNumber.F_BEGIN_FUNCTION OR	
				mOtherPosition.ZoneNumber > 0) AND 
				mOtherPosition.eFunctionNumber <> Position.eFunctionNumber THEN
					// Error: Index found on another location
					mReturnCode := E_ErrorConv.INDEX_MATCH_WITH_POSITION;
					// debug message: '11-000-0000-00-0,  data index found on another location,  telegram = TTA,  position = 99-999-9999-99-9,  TU_DataIndex = 3,  TuID = 012345,  AssignmentID = 87654321'
					DebugMsg:= '';
					DebugMsg:= CONCAT(DebugMsg, F_AddDividerToSisString(mpTTA^.Position));
					DebugMsg:= CONCAT(DebugMsg, ',  data index found on another location');
					DebugMsg:= CONCAT(DebugMsg, DebugTextBlocks.TELEGRAM);
					DebugMsg:= CONCAT(DebugMsg, 'TTA');
					DebugMsg:= CONCAT(DebugMsg, DebugTextBlocks.POSITION);
					DebugMsg:= CONCAT(DebugMsg, F_AddDividerToSisString(mOtherPosition.PositionName));
					DebugMsg:= CONCAT(DebugMsg, F_CreateTU_DataString(TU_DataIndex:= mTU_DataIndex));
					fbDebugMsg.M_SendErrorMsg(mMessage := DebugMsg);
	
					FCQ.Code:= E_ITC_FunctionControlCode.SET_ERROR;
					FCQ.Variable := INT_TO_DINT(mReturnCode);
					
					// Set corresponding position to error
					M_ProcessToFunction(
					meFunctionNumber	:= Position.eFunctionNumber,
					meChannelSrc		:= meChannelSrc,
					mMsgType			:= E_ITC_MsgTypeConv.FUNCTION_CONTROL_REQUEST,
					mpData				:= ADR(FCQ),
					mLen				:= SIZEOF(FCQ));
					
					M_ProcessToFunction(
					meFunctionNumber	:= mOtherPosition.eFunctionNumber,
					meChannelSrc		:= meChannelSrc,
					mMsgType			:= E_ITC_MsgTypeConv.FUNCTION_CONTROL_REQUEST,
					mpData				:= ADR(FCQ),
					mLen				:= SIZEOF(FCQ));
				END_IF
			END_IF
	
		// If the corresponding position consists of an empty TU-Data set, use that one
		ELSIF mTU_DataIndexPosition > 0 THEN
			mTU_DataIndex := mTU_DataIndexPosition;
		ELSE
			// Try insert TU-Data
			mTU_DataIndex := F_InsertTU_Data(
								eFunctionNumber := Position.eFunctionNumber,
								ZoneNumber 		:= Position.ZoneNumber);
			
			// No free TU Index was found
			IF mTU_DataIndex = 0 THEN
				// Error: No free TU-DataIndex
				mReturnCode := E_ErrorConv.NO_FREE_TU_DATA_SET;
				// debug message: '11-000-0000-00-0,  no free data index,  telegram = TTA,  TuID = 012345,  AssignmentID = 87654321'
				DebugMsg:= '';
				DebugMsg:= CONCAT(DebugMsg, F_AddDividerToSisString(mpTTA^.Position));
				DebugMsg:= CONCAT(DebugMsg, ',  no free data index');
				DebugMsg:= CONCAT(DebugMsg, DebugTextBlocks.TELEGRAM);
				DebugMsg:= CONCAT(DebugMsg, 'TTA');
				DebugMsg:= CONCAT(DebugMsg, DebugTextBlocks.TUID);
				DebugMsg:= CONCAT(DebugMsg, mpTTA^.TU_ID);
				DebugMsg:= CONCAT(DebugMsg, DebugTextBlocks.ASSIGNMENTID);
				DebugMsg:= CONCAT(DebugMsg, UDINT_TO_STRING(mpTTA^.AssignmentID) );
				fbDebugMsg.M_SendErrorMsg(mMessage := DebugMsg);
			END_IF
		END_IF
	END_IF
END_IF


(**************************************************************************************
already an error -> cancel processing
***************************************************************************************)
IF mReturnCode <> 0 THEN
	TTC.Position    := mpTTA^.Position;
	TTC.TU_DataIndex:= mTU_DataIndex;
	TTC.MsgSequence := mpTTA^.MsgSequence;
	TTC.TU_ID       := mpTTA^.TU_ID;
	TTC.AssignmentID:= mpTTA^.AssignmentID;
	TTC.ReturnCode  := mReturnCode;
	M_SendData(meChannel:= meChannelSrc, 
	mMsgType := E_ITC_MsgTypeConv.TRANSPORT_TASK_COMPLETE, 
	mpData   := ADR(TTC),
	mLen     := SIZEOF(TTC));
	// debug message already sent
	RETURN;
END_IF


(**************************************************************************************
If no TU_DataIndex is available
***************************************************************************************)
IF mTU_DataIndex <= 0 THEN
	RETURN;  // debug message already sent
END_IF


(**************************************************************************************
Update TU data -> process TTA
***************************************************************************************)
// Fill in the received TU-Data 
TU_DataTable[mTU_DataIndex].DataSet.DataPresent := TRUE;
TU_DataTable[mTU_DataIndex].DataSet.JobPresent  := FALSE;

IF mTU_ID_Present THEN
	TU_DataTable[mTU_DataIndex].TU_ID.HashCode := F_CreateHashCode(mpTTA^.TU_ID);
	TU_DataTable[mTU_DataIndex].TU_ID.ASCII    := mpTTA^.TU_ID;
ELSE
	TU_DataTable[mTU_DataIndex].TU_ID.HashCode := F_CreateHashCode(Conveyor.TU_ID_UNKNOWN);
	TU_DataTable[mTU_DataIndex].TU_ID.ASCII    := Conveyor.TU_ID_UNKNOWN;
END_IF

IF mAssignmentID_Present THEN
	TU_DataTable[mTU_DataIndex].AssignmentID := mpTTA^.AssignmentID;
ELSE
	TU_DataTable[mTU_DataIndex].AssignmentID := Conveyor.ASSIGNMENT_ID_UNKNOWN;
END_IF

TU_DataTable[mTU_DataIndex].DataSet.Dimension.Height:= mpTTA^.Height;
TU_DataTable[mTU_DataIndex].DataSet.Dimension.Length:= mpTTA^.Length;
TU_DataTable[mTU_DataIndex].DataSet.Dimension.Weight:= mpTTA^.Weight;
TU_DataTable[mTU_DataIndex].DataSet.Dimension.Width := mpTTA^.Width;
TU_DataTable[mTU_DataIndex].DataSet.Orientation		:= mpTTA^.Orientation;
TU_DataTable[mTU_DataIndex].DataSet.TU_Parameter	:= mpTTA^.TU_Parameter;
TU_DataTable[mTU_DataIndex].DataSet.TU_Type 		:= mpTTA^.TU_Type;
TU_DataTable[mTU_DataIndex].DataSet.IO_Data 		:= mpTTA^.IO_Data;
TU_DataTable[mTU_DataIndex].DataSet.LowerLimit 		:= mpTTA^.LowerLimit;
TU_DataTable[mTU_DataIndex].DataSet.UpperLimit 		:= mpTTA^.UpperLimit;
TU_DataTable[mTU_DataIndex].DataSet.Sequence 		:= mpTTA^.Sequence;			
TU_DataTable[mTU_DataIndex].DataSet.SubSequence 	:= mpTTA^.SubSequence;			
TU_DataTable[mTU_DataIndex].DataSet.SequenceSize 	:= mpTTA^.SequenceSize;		
TU_DataTable[mTU_DataIndex].DataSet.GroupID 		:= mpTTA^.GroupID;			
TU_DataTable[mTU_DataIndex].DataSet.GroupSize 		:= mpTTA^.GroupSize;	
TU_DataTable[mTU_DataIndex].DataSet.DestinationSlot := mpTTA^.DestinationSlot;	
TU_DataTable[mTU_DataIndex].DataSet.NumberOfDest	:= mpTTA^.NumberOfDestinations;

// Clear destination table 
MEMSET(destAddr := ADR(TU_DataTable[mTU_DataIndex].Destination), fillByte := 0, n := SIZEOF(TU_DataTable[mTU_DataIndex].Destination));


// debug message: '11-000-0000-00-0,  new destination assigned,  telegram = TTA,  TU_DataIndex = 3,  TuID = 123456,  AssignmentID = 87654321,  destination = 99-999-9999-99-9,  destination = 99-999-9999-99-9'
DebugMsg:= '';
DebugMsg:= CONCAT(DebugMsg, F_AddDividerToSisString(mpTTA^.Position));
DebugMsg:= CONCAT(DebugMsg, ',  new destination assigned');
DebugMsg:= CONCAT(DebugMsg, DebugTextBlocks.TELEGRAM);
DebugMsg:= CONCAT(DebugMsg, 'TTA');
IF NOT mRequestForPosition THEN
	mOtherPosition:= F_SearchPositionOfTU_Index(TU_DataIndex        := mTU_DataIndex,
	eStartFunctionNumber:= F_BEGIN_FUNCTION);
	DebugMsg:= CONCAT(DebugMsg, DebugTextBlocks.POSITION);
	DebugMsg:= CONCAT(DebugMsg, F_AddDividerToSisString(mOtherPosition.PositionName));
END_IF
DebugMsg:= CONCAT(DebugMsg, F_CreateTU_DataString(TU_DataIndex:= mTU_DataIndex));

// Fill in the destinations 
mDestIndex := 1;
FOR Idx := 1 TO mpTTA^.NumberOfDestinations DO
	// Destination was found 
	IF mDestinationPosition[Idx].eFunctionNumber <> E_FunctionNumber.F_BEGIN_FUNCTION THEN
		TU_DataTable[mTU_DataIndex].DataSet.JobPresent := TRUE;
		TU_DataTable[mTU_DataIndex].Destination[mDestIndex].eFunctionNumber := mDestinationPosition[Idx].eFunctionNumber;
		TU_DataTable[mTU_DataIndex].Destination[mDestIndex].ZoneNumber 		:= mDestinationPosition[Idx].ZoneNumber;
		TU_DataTable[mTU_DataIndex].Destination[mDestIndex].PositionName	:= mpTTA^.Destination[Idx];
		// debug message
		DebugMsg:= CONCAT(DebugMsg, DebugTextBlocks.DESTINATION);
		DebugMsg:= CONCAT(DebugMsg, F_AddDividerToSisString(mpTTA^.Destination[Idx]));
		// continue
		mDestIndex := mDestIndex + 1;
	ELSE
		// Check if it's an external destination
		IF mVirtualDestinationPosition[Idx].eFunctionNumber <> E_FunctionNumber.F_BEGIN_VIRTUAL_FUNCTION THEN
			TU_DataTable[mTU_DataIndex].DataSet.JobPresent := TRUE;
			TU_DataTable[mTU_DataIndex].Destination[mDestIndex].eFunctionNumber 	:= mVirtualDestinationPosition[Idx].eFunctionNumber;
			TU_DataTable[mTU_DataIndex].Destination[mDestIndex].ZoneNumber 			:= 0;
			TU_DataTable[mTU_DataIndex].Destination[mDestIndex].PositionName		:= mpTTA^.Destination[Idx];
			// debug message
			DebugMsg:= CONCAT(DebugMsg, DebugTextBlocks.DESTINATION);
			DebugMsg:= CONCAT(DebugMsg, F_AddDividerToSisString(mpTTA^.Destination[Idx]));
			// continue
			mDestIndex := mDestIndex + 1;
		END_IF
	END_IF
END_FOR

// fire debug message only when if destination exists
IF mDestIndex <> 0 THEN
	fbDebugMsg.M_SendInfoMsg(mMessage := DebugMsg);
END_IF


// Update time stamp 
TU_DataTable[mTU_DataIndex].TimeStamp.eInsertFunctionNumber := E_FunctionNumber.F_BEGIN_FUNCTION;
TU_DataTable[mTU_DataIndex].TimeStamp.InsertZoneNumber := 0;
TU_DataTable[mTU_DataIndex].TimeStamp.InsertDateTime       := System.fbSystemTime.TIMESTR;

// If TTA was sent to a Position 
IF mRequestForPosition THEN
	Data.Init := TRUE;
	Data.TU_DataIndex := mTU_DataIndex;
	Data.ZoneNumber := Position.ZoneNumber;
	
	// Forward to position
	M_ProcessToFunction(meFunctionNumber:= Position.eFunctionNumber, 
						meChannelSrc	:= meChannelSrc, 
						mMsgType		:= E_ITC_MsgTypeConv.ADD_TU_DATA,
						mpData			:= ADR(Data), 
						mLen			:= SIZEOF(Data));
	
	// Update TimeStamp position
	TU_DataTable[mTU_DataIndex].TimeStamp.eInsertFunctionNumber := Position.eFunctionNumber;
	TU_DataTable[mTU_DataIndex].TimeStamp.InsertZoneNumber		:= Position.ZoneNumber;
END_IF



(**************************************************************************************
If position number and zone index is identical  (position = destination)
***************************************************************************************)
// if TTA was send to subsystem -> use TUs position
IF NOT mRequestForPosition THEN
	Position:= mOtherPosition;
END_IF

IF F_DeleteDestination( eFunctionNumber := Position.eFunctionNumber, ZoneNumber := Position.ZoneNumber) THEN

	TTC.Position := mpTTA^.Position;
	TTC.TU_DataIndex := mTU_DataIndex;
	TTC.MsgSequence := mpTTA^.MsgSequence;
	TTC.TU_ID := mpTTA^.TU_ID;
	TTC.AssignmentID := mpTTA^.AssignmentID;
	TTC.ReturnCode := E_ErrorConv.NO_ERROR_CODE;
	
	M_SendData(meChannel:= meChannelSrc, 
	mMsgType := E_ITC_MsgTypeConv.TRANSPORT_TASK_COMPLETE, 
	mpData   := ADR(TTC),
	mLen	 := SIZEOF(TTC));
	
	// debug message: '11-000-0000-00-0,  destination and position are equal,  telegram = TTA'
	DebugMsg:= '';
	DebugMsg:= CONCAT(DebugMsg, F_AddDividerToSisString(mpTTA^.Position));
	DebugMsg:= CONCAT(DebugMsg, ',  destination and position are equal');
	DebugMsg:= CONCAT(DebugMsg, DebugTextBlocks.TELEGRAM);
	DebugMsg:= CONCAT(DebugMsg, 'TTA');
	IF NOT mRequestForPosition THEN
		DebugMsg:= CONCAT(DebugMsg, DebugTextBlocks.POSITION);
		DebugMsg:= CONCAT(DebugMsg, F_AddDividerToSisString(Position.PositionName));
	END_IF
	
	fbDebugMsg.M_SendErrorMsg(mMessage := DebugMsg);
END_IF
END_METHOD

METHOD PROTECTED M_ProcessTUQ : BOOL
(**************************************************************************************
 * 	Application		:	BoxControl Framework
 *	Revision		:	$Revision: 474929 $
 *	Revision date	:	$Date: 2021-04-08 12:45:11 +0200 (tor, 08 apr 2021) $
 *	Last changed by	:	$Author: b7gessa $
 *	URL				:	$URL: http://almscdc.swisslog.com/repo/SWPD/Development/BoxControlFramework/20_Release/tags/R1.12.0/01_Software/BCF/BCF/JumpStart/20_Product/10_BCF/11_Conv/11_Com/11_ITC/FB_ITC_Conveyor.TcPOU $
 *
 *	Purpose			:	Process a received Transport Unit Request telegram.
 *
 * ------------------------------------------------------------------------------------
 *	Copyright Swisslog [IP AG], Switzerland. All rights reserved.
 * 
 * ------------------------------------------------------------------------------------
 *	
 * 	Revision History: 
 *
 * 	VERSION			DATE			INITIALS			DESCRIPTION
 *	0.1				01.01.2001		swl					Example
 *
 **************************************************************************************)
 VAR_INPUT
	meChannelSrc		: E_MFCS_Channel; // Source communicaton channel
	mpTUQ				: POINTER TO ST_ITC_TUQ; // Pointer to TTA
	mLen				: UDINT; // Data length
END_VAR

VAR
	mTU_DataIndex		: DINT; // TU_DataIndex from zone
	mErrorCode			: E_ErrorConv; // ErrorCode
	mPositionName		: STRING(Conveyor.POSITION_STRINGLENGTH); // SIS Position name MM-000-0000-000
	mDestination		: ARRAY [1..Conveyor.NUMBER_OF_DESTINATIONS] OF STRING(Conveyor.POSITION_STRINGLENGTH); // Array of 12 Digit SIS Destinations
	mDestinationIndex	: INT; // DestinationIndex
	mName				: STRING; // temp name
END_VAR
// Initialize
M_ProcessTUQ := TRUE;

// Search TU_DataIndex in the TU-DataTable
mTU_DataIndex := F_SearchTU_ByHashCode(TU_ID := mpTUQ^.TU_ID);

// If TU-ID was found
IF mTU_DataIndex <> 0 THEN
	
	// Get Destinations
	FOR mDestinationIndex := 1 TO TU_DataTable[mTU_DataIndex].DataSet.NumberOfDest DO
		mName := F_GetFunctionName( 
					eFunctionNumber := TU_DataTable[mTU_DataIndex].Destination[mDestinationIndex].eFunctionNumber,
					ZoneNumber		:= TU_DataTable[mTU_DataIndex].Destination[mDestinationIndex].ZoneNumber);
												
		mDestination[mDestinationIndex] := F_ReduceToAlphaNumeric(InputString := mName);
	END_FOR
	
	// Get PositionName from TU_Data
	mPositionName := F_GetFunctionName(
						eFunctionNumber := TU_DataTable[mTU_DataIndex].TimeStamp.eInsertFunctionNumber,
						ZoneNumber		:= 0);
	
	TUR.Position := F_ReduceToAlphaNumeric(InputString := mPositionName);
	TUR.TU_DataIndex := mTU_DataIndex;
	TUR.TU_ID := TU_DataTable[mTU_DataIndex].TU_ID.ASCII;
	TUR.TU_Type := TU_DataTable[mTU_DataIndex].DataSet.TU_Type;
	TUR.AssignmentID := TU_DataTable[mTU_DataIndex].AssignmentID;
	TUR.Length := TU_DataTable[mTU_DataIndex].DataSet.Dimension.Length;
	TUR.Width := TU_DataTable[mTU_DataIndex].DataSet.Dimension.Width;
	TUR.Height := TU_DataTable[mTU_DataIndex].DataSet.Dimension.Height;
	TUR.Weight := TU_DataTable[mTU_DataIndex].DataSet.Dimension.Weight;
	TUR.Orientation := TU_DataTable[mTU_DataIndex].DataSet.Orientation;
	TUR.TU_Parameter := TU_DataTable[mTU_DataIndex].DataSet.TU_Parameter;
	TUR.IO_Data := TU_DataTable[mTU_DataIndex].DataSet.IO_Data;
	TUR.LowerLimit := TU_DataTable[mTU_DataIndex].DataSet.LowerLimit;
	TUR.UpperLimit := TU_DataTable[mTU_DataIndex].DataSet.UpperLimit;
	TUR.Sequence :=	TU_DataTable[mTU_DataIndex].DataSet.Sequence;			
	TUR.SubSequence := TU_DataTable[mTU_DataIndex].DataSet.SubSequence;			
	TUR.SequenceSize :=	TU_DataTable[mTU_DataIndex].DataSet.SequenceSize;		
	TUR.GroupID := TU_DataTable[mTU_DataIndex].DataSet.GroupID;			
	TUR.GroupSize := TU_DataTable[mTU_DataIndex].DataSet.GroupSize;	
	TUR.DestinationSlot :=TU_DataTable[mTU_DataIndex].DataSet.DestinationSlot;		
	TUR.ReturnCode := E_ErrorConv.NO_ERROR_CODE;
	TUR.NumberOfDestinations := TU_DataTable[mTU_DataIndex].DataSet.NumberOfDest;
	TUR.Destination := mDestination;
	
	M_SendData(
		meChannel := meChannelSrc, 
		mMsgType  := E_ITC_MsgTypeConv.TRANSPORT_UNIT_REPORT, 
		mpData    := ADR(TUR),
		mLen	  := SIZEOF(TUR));		
				
ELSE
	TUR.Position := '';
	TUR.TU_DataIndex := 0;
	TUR.TU_ID := mpTUQ^.TU_ID;
	TUR.TU_Type := 0;
	TUR.AssignmentID := 0;
	TUR.Length := 0;
	TUR.Width := 0;
	TUR.Height := 0;
	TUR.Weight := 0;
	TUR.Orientation := '   ';
	TUR.TU_Parameter := 0;
	TUR.IO_Data := 0;
	TUR.LowerLimit := 0;
	TUR.UpperLimit := 0;
	TUR.Sequence :=	0;			
	TUR.SubSequence := 0;			
	TUR.SequenceSize :=	0;		
	TUR.GroupID := 0;			
	TUR.GroupSize := 0;	
	TUR.DestinationSlot :=	0;			
	TUR.ReturnCode := E_ErrorConv.TU_ID_WRONG;
	TUR.NumberOfDestinations := 0;
	TUR.Destination := mDestination;
	
	M_SendData(
		meChannel := meChannelSrc, 
		mMsgType  := E_ITC_MsgTypeConv.TRANSPORT_UNIT_REPORT, 
		mpData    := ADR(TUR),
		mLen	  := SIZEOF(TUR));	
END_IF
END_METHOD

METHOD M_ProcessVIQ : BOOL
(**************************************************************************************
 * 	Application		:	BoxControl Framework
 *	Revision		:	$Revision: 474929 $
 *	Revision date	:	$Date: 2021-04-08 12:45:11 +0200 (tor, 08 apr 2021) $
 *	Last changed by	:	$Author: b7gessa $
 *	URL				:	$URL: http://almscdc.swisslog.com/repo/SWPD/Development/BoxControlFramework/20_Release/tags/R1.12.0/01_Software/BCF/BCF/JumpStart/20_Product/10_BCF/11_Conv/11_Com/11_ITC/FB_ITC_Conveyor.TcPOU $
 *
 *	Purpose			:	Process a received Transport Task Assignment telegram.
 *
 * ------------------------------------------------------------------------------------
 *	Copyright Swisslog [IP AG], Switzerland. All rights reserved.
 * 
 * ------------------------------------------------------------------------------------
 *	
 * 	Revision History: 
 *
 * 	VERSION			DATE			INITIALS			DESCRIPTION
 *	0.1				10.03.2016		Kay Röder			Example
 *
 **************************************************************************************)
VAR_INPUT
	meChannelSrc					: E_MFCS_Channel; // Source communication channel
	mpVIQ							: POINTER TO ST_ITC_VIQ; // Pointer to VIQ
	mLen							: UDINT;
END_VAR
VAR
	meFunctionPosition			: ST_PositionIdent; // Position
	meGroupNumber				: E_GroupNumber; // Group
	meElementNumber				: E_ElementNumber;//Element Number
	meSubsystem					: BOOL;	//Subsystem
	mKeyValuePairs				: ARRAY [1..System.NUMBER_OF_KEYVALUE_PAIRS_VIR] OF ST_ITC_VIR_SET;
END_VAR
// Initialize
M_ProcessVIQ := TRUE;

// Get position from message
meFunctionPosition := F_SearchFunctionPosition(Position := mpVIQ^.Position);
meElementNumber    := F_SearchElementPosition(ElementName := mpVIQ^.Position);
meGroupNumber      := F_SearchGroupNumber(GroupName := mpVIQ^.Position);
meSubsystem 	   := F_EqualSisNames(Name1 := SubsystemRegistry.SubSystemName,
                                    Name2 := mpVIQ^.Position);
														
// If a valid function was found with a valid zone
IF 	meFunctionPosition.eFunctionNumber > E_FunctionNumber.F_BEGIN_FUNCTION AND 
	meFunctionPosition.eFunctionNumber < E_FunctionNumber.F_END_FUNCTION AND 
	meFunctionPosition.ZoneNumber >= 0 AND meFunctionPosition.ZoneNumber <= NUMBER_OF_ZONES_PER_FUNCTION THEN
	
	// Forward to function
	M_ProcessVIQ := M_ProcessToFunction(
						meFunctionNumber	:= meFunctionPosition.eFunctionNumber, 
						meChannelSrc		:= meChannelSrc, 
						mMsgType			:= E_ITC_MsgTypeConv.VISUALIZATION_INFORMATION_REQUEST,
						mpData				:= mpVIQ,
						mLen				:= mLen);

// If a valid element was found
ELSIF meElementNumber > E_ElementNumber.E_BEGIN_ELEMENT AND
 	  meElementNumber < E_ElementNumber.E_END_ELEMENT THEN

	// Forward to element
	M_ProcessVIQ := M_ProcessToElement(
						meElementNumber		:= meElementNumber, 
						meChannelSrc		:= meChannelSrc, 
						mMsgType			:= E_ITC_MsgTypeConv.VISUALIZATION_INFORMATION_REQUEST,
						mpData				:= mpVIQ,
						mLen				:= mLen);	

// If a valid group was found
ELSIF meGroupNumber > E_GroupNumber.G_BEGIN_GROUP AND
 	  meGroupNumber < E_GroupNumber.G_END_GROUP THEN

	// Forward to group
	M_ProcessVIQ := M_ProcessToGroup(
						meGroupNumber		:= meGroupNumber, 
						meChannelSrc		:= meChannelSrc, 
						mMsgType			:= E_ITC_MsgTypeConv.VISUALIZATION_INFORMATION_REQUEST,
						mpData				:= mpVIQ,
						mLen				:= mLen);		

// If a valid subsystem was found
ELSIF meSubsystem THEN

	// Forward to subsystem
	M_ProcessVIQ := M_ProcessToSubsystem(
						meChannelSrc		:= meChannelSrc, 
						mMsgType			:= E_ITC_MsgTypeConv.VISUALIZATION_INFORMATION_REQUEST,
						mpData				:= mpVIQ,
						mLen				:= mLen);	
ELSE
	// Unknown Position name received 
	DebugMsg := CONCAT('VIQ: Unknown address', mpVIQ^.Position);
	fbDebugMsg.M_SendErrorMsg(mMessage := DebugMsg); 
	
	// Send VIR - error - no valid Address
	F_ITC_SendVIR(
		eChannelSrc := meChannelSrc,
		Position := mpVIQ^.Position,
		NumOfKeyValuePairs := 1,
		KeyValuePairs	:= mKeyValuePairs);
END_IF
END_METHOD

METHOD M_SendData : BOOL
(**************************************************************************************
 * 	Application		:	BoxControl Framework
 *	Revision		:	$Revision: 474929 $
 *	Revision date	:	$Date: 2021-04-08 12:45:11 +0200 (tor, 08 apr 2021) $
 *	Last changed by	:	$Author: b7gessa $
 *	URL				:	$URL: http://almscdc.swisslog.com/repo/SWPD/Development/BoxControlFramework/20_Release/tags/R1.12.0/01_Software/BCF/BCF/JumpStart/20_Product/10_BCF/11_Conv/11_Com/11_ITC/FB_ITC_Conveyor.TcPOU $
 *
 *	Purpose			:	Send data to MFCS connection
 *
 * ------------------------------------------------------------------------------------
 *	Copyright Swisslog [IP AG], Switzerland. All rights reserved.
 * 
 * ------------------------------------------------------------------------------------
 *	
 * 	Revision History: 
 *
 * 	VERSION			DATE			INITIALS			DESCRIPTION
 *	0.1				01.01.2001		swl					Example
 *
 **************************************************************************************)
VAR_INPUT
	meChannel				: E_MFCS_Channel; // Channel to forward msg
	mMsgType				: INT; // Msg type
	mpData					: PVOID; // Data pointer
	mLen					: UDINT; // Data length
END_VAR

VAR
	mMFCS_Instance			: ITF_MFCS; // Instance to compare valid interfaces
END_VAR
// INitialize
M_SendData := TRUE;

// If communication with single source
IF meChannel <> 0 THEN
	IF __QUERYINTERFACE(fbMFCS_Channel[meChannel], mMFCS_Instance) THEN
		// Forward data to MFCS channel
		M_SendData := fbMFCS_Channel[meChannel].M_SendData(
						meChannelSrc := meChannel,
						mMsgType  	 := mMsgType,
						mpData	  	 := mpData,
						mLen		 := mLen);
	END_IF			
// Sender unknown - forward to all
ELSE
	FOR Idx := E_MFCS_Channel.BEGIN_CHANNEL + 1 TO E_MFCS_Channel.END_CHANNEL - 1 DO
		IF __QUERYINTERFACE(fbMFCS_Channel[Idx], mMFCS_Instance) THEN
			// Forward data to MFCS channel
			fbMFCS_Channel[Idx].M_SendData(
				meChannelSrc := meChannel,
				mMsgType  	 := mMsgType,
				mpData	  	 := mpData,
				mLen		 := mLen);
		END_IF
	END_FOR
END_IF
END_METHOD

END_FUNCTION_BLOCK

// ---- 20_Product/10_BCF/11_Conv/11_Com/11_ITC/F_ITC_SendSDI.TcPOU
FUNCTION F_ITC_SendSDI : BOOL
(**************************************************************************************
 * 	Application		:	BoxControl Framework
 *	Revision		:	$Revision: 404529 $
 *	Revision date	:	$Date: 2018-04-23 08:21:38 +0200 (Mo., 23 Apr 2018) $
 *	Last changed by	:	$Author: b7bolm $
 *	URL				:	$URL: http://almscdc.swisslog.com/repo/SWPD/Development/BoxControlFramework/20_Release/trunk/01_Software/BCF/BCF/JumpStart/20_Product/10_App/11_Com/10_Lib/10_Conv/11_ITC/F_ITC_SendSDI.TcPOU $
 *
 *	Purpose			:	Wrap message - SIR
 *
 * ------------------------------------------------------------------------------------
 *	Copyright Swisslog [IP AG], Switzerland. All rights reserved.
 * 
 * ------------------------------------------------------------------------------------
 *	
 * 	Revision History: 
 *
 * 	VERSION			DATE			INITIALS			DESCRIPTION
 *	0.1				01.01.2001		swl					Example
 *
 **************************************************************************************)
VAR_INPUT
	eChannelSrc		: E_MFCS_Channel; // Source communicaton channel	
	SignalNumber	: INT; // Signal Number
	SignalState		: BOOL; // Signal Status
	eReturnCode		: E_ErrorConv; // Return code
END_VAR
VAR
	SDI				: ST_ITC_SDI; 
END_VAR

// Map values
SDI.SignalState := SignalState;
SDI.SignalNumber := SignalNumber;
SDI.ReturnCode := eReturnCode;

// Forward to ITC
F_ITC_SendSDI := fbITC_Manager.M_SendData(
					meChannel	:= eChannelSrc,
					mMsgType	:= E_ITC_MsgTypeConv.SEND_DIGITAL_INPUT,
					mpData		:= ADR(SDI),
					mLen		:= SIZEOF(SDI));

END_FUNCTION

// ---- 20_Product/10_BCF/11_Conv/12_E_Functions/10_Helper/F_SearchFunctionPosition.TcPOU
FUNCTION F_SearchFunctionPosition : ST_PositionIdent
(**************************************************************************************
 * 	Application		:	BoxControl Framework
 *	Revision		:	$Revision: 404529 $
 *	Revision date	:	$Date: 2018-04-23 08:21:38 +0200 (Mo., 23 Apr 2018) $
 *	Last changed by	:	$Author: b7bolm $
 *	URL				:	$URL: http://almscdc.swisslog.com/repo/SWPD/Development/BoxControlFramework/20_Release/trunk/01_Software/BCF/BCF/JumpStart/20_Product/10_App/12_E_Functions/10_Lib/10_Conv/10_Functions/F_SearchFunctionPosition.TcPOU $
 *
 *	Purpose			:	Search a position in the function registry.
 *
 * ------------------------------------------------------------------------------------
 *	Copyright Swisslog [IP AG], Switzerland. All rights reserved.
 * 
 * ------------------------------------------------------------------------------------
 *	
 * 	Revision History: 
 *
 * 	VERSION			DATE			INITIALS			DESCRIPTION
 *	0.1				01.01.2001		swl					Example
 *
 **************************************************************************************)
VAR_INPUT
	Position			: STRING(NAME_LENGTH); // Name of position
END_VAR

VAR
	NameHashCode		: UDINT; // Name converted to hash code
	eFunctionNumber		: E_FunctionNumber; // Function number
	ZoneNumber			: INT; // Zone number
END_VAR

// Initialize
F_SearchFunctionPosition.eFunctionNumber := E_FunctionNumber.F_BEGIN_FUNCTION;
F_SearchFunctionPosition.ZoneNumber		 := 0;

// Build Hash code
NameHashCode := F_CreateHashCode(InputString := Position);

// Loop trough function registry
FOR eFunctionNumber := E_FunctionNumber.F_BEGIN_FUNCTION + 1 TO E_FunctionNumber.F_END_FUNCTION - 1 DO	
	// Compare Hash code of function
	IF FunctionRegistry[eFunctionNumber].HashCode = NameHashCode THEN
		// Compare String name	
		IF F_EqualSisNames(Name1 := FunctionRegistry[eFunctionNumber].FunctionName,
                       Name2 := Position) THEN
			// Function found - return
			F_SearchFunctionPosition.eFunctionNumber := eFunctionNumber;
			F_SearchFunctionPosition.ZoneNumber		 := 0;
			F_SearchFunctionPosition.PositionName    := Position;
			RETURN;
		END_IF
	END_IF

	// Compare Hash code of zones
	FOR ZoneNumber := 1 TO F_GetNumberOfZones(eFunctionNumber := eFunctionNumber) DO
		// If zone number is within the limit
		IF ZoneNumber <= NUMBER_OF_ZONES_PER_FUNCTION THEN 
			// Compare Hash code of zone
			IF FunctionRegistry[eFunctionNumber].Zone[ZoneNumber].HashCode = NameHashCode THEN
				// Compare String name	
				IF F_EqualSisNames(Name1 := FunctionRegistry[eFunctionNumber].Zone[ZoneNumber].ZoneName,
                           Name2 := Position) THEN
					// Zone found - return
					F_SearchFunctionPosition.eFunctionNumber := eFunctionNumber;
					F_SearchFunctionPosition.ZoneNumber		 := ZoneNumber;
					F_SearchFunctionPosition.PositionName    := Position;
					RETURN;
				END_IF
			END_IF
		ELSE
			EXIT;
		END_IF	
	END_FOR
END_FOR

// When nothing was found, try virtual destinations
F_SearchFunctionPosition := F_GetVirtualDestination(Position);

END_FUNCTION

// ---- 20_Product/10_BCF/11_Conv/12_E_Functions/10_Helper/F_EqualSisNames.TcPOU
// compares two sis names, all characters (except numbers and letters) will be ignored
FUNCTION PUBLIC F_EqualSisNames : BOOL

(**************************************************************************************
 * Application   : BoxControl Framework
 * Revision date : $Date: 2013-09-23 11:26:06 +0200 (Wed, 23 Sep 2015) $
 * Author        : CDC
 * ------------------------------------------------------------------------------------
 * © Swisslog AG * Swisslog is not liable for any usage of this source code that is not agreed
 * on between Swisslog and the other party. The mandatory legal liability remains * unaffected.
 * ------------------------------------------------------------------------------------
 * Project revision history:
 *
 * VERSION DATE         INITIALS     DESCRIPTION
 * 0.0     DD.MM.YYYY   (name)       (explain customized modifications)
 *
 **************************************************************************************)

//***********************************************************************************************************
VAR_INPUT
  Name1                 : STRING[NAME_LENGTH]         := '';
  Name2                 : STRING[NAME_LENGTH]         := '';
END_VAR

//***********************************************************************************************************
VAR
  Idx1                  : WORD                        := 0;
  Idx2                  : WORD                        := 0;
END_VAR


//***********************************************************************************************************
//** check each character ***********************************************************************************
Idx1:= 0;
Idx2:= 0;

WHILE TRUE DO
	//-- seek next number @ Name1 ---------------------------------------------------------
	WHILE Name1[Idx1] <> 16#00 DO	// hint: AND connects stronger than OR, but brackets are not recommended by coding "guidelines"
		//-- is number/letter -> stopp --------------
		IF(Name1[Idx1] >= 16#30)AND(Name1[Idx1] <= 16#39)       // 0..9
		OR(Name1[Idx1] >= 16#41)AND(Name1[Idx1] <= 16#5A)       // A..Z
		OR(Name1[Idx1] >= 16#61)AND(Name1[Idx1] <= 16#7A) THEN  // a..z
			EXIT;
		END_IF
		//-- continue -------------------------------
		Idx1:= Idx1 + 1;
	END_WHILE

	//-- seek next number @ Name2 ---------------------------------------------------------
	WHILE Name2[Idx2] <> 16#00 DO	// hint: AND connects stronger than OR, but brackets are not recommended by coding "guidelines"
		//-- is number/letter -> stopp --------------
		IF (Name2[Idx2] >= 16#30)AND(Name2[Idx2] <= 16#39)      // 0..9
		 OR(Name2[Idx2] >= 16#41)AND(Name2[Idx2] <= 16#5A)      // A..Z
		 OR(Name2[Idx2] >= 16#61)AND(Name2[Idx2] <= 16#7A) THEN // a..z

			EXIT;
		END_IF
		//-- continue -------------------------------
		Idx2:= Idx2 + 1;
	END_WHILE

	//-- both names end here toghether ----------------------------------------------------
	IF Name1[Idx1] = 16#00 AND Name2[Idx2] = 16#00 THEN
		EXIT;

	//-- one of the names end here --------------------------------------------------------
	ELSIF Name1[Idx1] = 16#00 OR Name2[Idx2] = 16#00 THEN
		F_EqualSisNames:= FALSE;
		RETURN;

	//-- compare --------------------------------------------------------------------------
	ELSIF Name1[Idx1] <> Name2[Idx2] THEN
		F_EqualSisNames:= FALSE;
		RETURN;
	END_IF

	// next characters --------------------------------------------------------------------
	Idx1:= Idx1 + 1;
	Idx2:= Idx2 + 1;

END_WHILE




//***********************************************************************************************************
//** done ***************************************************************************************************
F_EqualSisNames:= TRUE;

END_FUNCTION

// ---- 20_Product/10_BCF/11_Conv/10_Base/F_GetVirtualDestination.TcPOU
FUNCTION F_GetVirtualDestination : ST_PositionIdent
(**************************************************************************************
 * 	Application		:	BoxControl Framework
 *	Revision		:	$Revision: 404529 $
 *	Revision date	:	$Date: 2018-04-23 08:21:38 +0200 (Mo., 23 Apr 2018) $
 *	Last changed by	:	$Author: b7bolm $
 *	URL				:	$URL: http://almscdc.swisslog.com/repo/SWPD/Development/BoxControlFramework/20_Release/trunk/01_Software/BCF/BCF/JumpStart/20_Product/10_App/10_Base/10_Lib/10_Conv/F_GetVirtualDestination.TcPOU $
 *
 *	Purpose			:	Returns virtual function number of an external destination.
 *
 * ------------------------------------------------------------------------------------
 *	Copyright Swisslog [IP AG], Switzerland. All rights reserved.
 * 
 * ------------------------------------------------------------------------------------
 *	
 * 	Revision History: 
 *
 * 	VERSION			DATE			INITIALS			DESCRIPTION
 *	0.1				26.07.2017		swl					Example
 *
 **************************************************************************************)
VAR_INPUT
	PositionName		: STRING(NAME_LENGTH); // Name of position
END_VAR

VAR
	eFunctionNumber		: E_FunctionNumber;
	HashCode			: UDINT;
	Idx					: INT;
	DestinationFound	: BOOL;
END_VAR

// Initialize
F_GetVirtualDestination.eFunctionNumber := E_FunctionNumber.F_BEGIN_FUNCTION;
F_GetVirtualDestination.PositionName := '';
F_GetVirtualDestination.ZoneNumber := 0;
DestinationFound := FALSE;

// Get hash code
HashCode := F_CreateHashCode(PositionName);

// Search virtual destination which belongs to this external destination
FOR eFunctionNumber := F_BEGIN_VIRTUAL_FUNCTION + 1 TO F_END_VIRTUAL_FUNCTION - 1 DO
	FOR Idx := 1 TO Conveyor.NUMBER_OF_EXT_DESTINATIONS DO
		// Compare hash code
		IF ExternalDestinationTable[eFunctionNumber, Idx].HashCode = HashCode THEN
			// Compare string name	
			IF F_EqualSisNames(Name1 := ExternalDestinationTable[eFunctionNumber, Idx].PositionName,
										     Name2 := PositionName) THEN
										
				F_GetVirtualDestination.eFunctionNumber := eFunctionNumber;
				F_GetVirtualDestination.PositionName := PositionName;
				F_GetVirtualDestination.ZoneNumber := 0;
				DestinationFound := TRUE;
				EXIT;
			END_IF
		END_IF
	END_FOR
	
	IF DestinationFound THEN
		EXIT;
	END_IF
END_FOR

END_FUNCTION

// ---- 20_Product/10_BCF/11_Conv/13_Elements/10_Helper/F_SearchElementPosition.TcPOU
FUNCTION F_SearchElementPosition : E_ElementNumber
(**************************************************************************************
 * 	Application		:	BoxControl Framework
 *	Revision		:	$Revision: 404529 $
 *	Revision date	:	$Date: 2018-04-23 08:21:38 +0200 (Mo., 23 Apr 2018) $
 *	Last changed by	:	$Author: b7bolm $
 *	URL				:	$URL: http://almscdc.swisslog.com/repo/SWPD/Development/BoxControlFramework/20_Release/trunk/01_Software/BCF/BCF/JumpStart/20_Product/10_App/13_Elements/10_Lib/10_Conv/10_Functions/F_SearchElementPosition.TcPOU $
 *
 *	Purpose			:	Search a position in the element registry.
 *
 * ------------------------------------------------------------------------------------
 *	Copyright Swisslog [IP AG], Switzerland. All rights reserved.
 * 
 * ------------------------------------------------------------------------------------
 *	
 * 	Revision History: 
 *
 * 	VERSION			DATE			INITIALS			DESCRIPTION
 *	0.1				01.01.2001		swl					Example
 *
 **************************************************************************************)
VAR_INPUT
	ElementName			: STRING(NAME_LENGTH); // Name of element
END_VAR

VAR
	NameHashCode		: UDINT; // Name converted to hash code
	eElementNumber		: E_ElementNumber; // Iterator
END_VAR


// Initialize
F_SearchElementPosition := E_ElementNumber.E_BEGIN_ELEMENT;

// Build Hash code
NameHashCode := F_CreateHashCode(InputString := ElementName);

// Loop over all groups 
FOR eElementNumber :=  E_ElementNumber.E_BEGIN_ELEMENT + 1 TO  E_ElementNumber.E_END_ELEMENT - 1 DO
	// Identical HashCode found 
	IF ElementRegistry[eElementNumber].HashCode = NameHashCode THEN
		// Element name is also identical 
		IF F_EqualSisNames(Name1:= ElementRegistry[eElementNumber].ElementName,
                       Name2:= ElementName) THEN	
				//Return element number
				F_SearchElementPosition := eElementNumber;
			RETURN;
		END_IF
	END_IF
END_FOR

END_FUNCTION

// ---- 20_Product/10_BCF/11_Conv/14_Groups/10_Helper/F_SearchGroupNumber.TcPOU
FUNCTION F_SearchGroupNumber : E_GroupNumber
(**************************************************************************************
 * 	Application		:	BoxControl Framework
 *	Revision		:	$Revision: 404529 $
 *	Revision date	:	$Date: 2018-04-23 08:21:38 +0200 (Mo., 23 Apr 2018) $
 *	Last changed by	:	$Author: b7bolm $
 *	URL				:	$URL: http://almscdc.swisslog.com/repo/SWPD/Development/BoxControlFramework/20_Release/trunk/01_Software/BCF/BCF/JumpStart/20_Product/10_App/14_Groups/10_Lib/10_Conv/10_Functions/F_SearchGroupNumber.TcPOU $
 *
 *	Purpose			:	Search a GroupNumber in the function registry.
 *
 * ------------------------------------------------------------------------------------
 *	Copyright Swisslog [IP AG], Switzerland. All rights reserved.
 * 
 * ------------------------------------------------------------------------------------
 *	
 * 	Revision History: 
 *
 * 	VERSION			DATE			INITIALS			DESCRIPTION
 *	0.1				01.01.2001		swl					Example
 *
 **************************************************************************************)
VAR_INPUT
	GroupName		:STRING(NAME_LENGTH); // GroupName as String
END_VAR

VAR
	NameHashCode  	:UDINT; // HashCode of the GroupName
	eGroupNumber	:E_GroupNumber; // Number of the group
END_VAR

// Initialize
F_SearchGroupNumber := E_GroupNumber.G_BEGIN_GROUP;

// Build Hash code
NameHashCode := F_CreateHashCode(InputString := GroupName);

// Loop over all groups 
FOR eGroupNumber :=  E_GroupNumber.G_BEGIN_GROUP + 1 TO  E_GroupNumber.G_END_GROUP - 1 DO
	// Identical HashCode found 
	IF GroupRegistry[eGroupNumber].HashCode = NameHashCode THEN
		// Group name is also identical 
		IF F_EqualSisNames(Name1 := GroupRegistry[eGroupNumber].GroupName,
                       Name2 := GroupName) THEN	
				//Return group number
				F_SearchGroupNumber := eGroupNumber;
			RETURN;
		END_IF
	END_IF
END_FOR

END_FUNCTION

// ---- 20_Product/10_BCF/11_Conv/12_E_Functions/10_Helper/F_FindFunction.TcPOU
// returns the function number of the functions name or F_BEGIN_FUNCTION if not found
FUNCTION PUBLIC F_FindFunction : E_FunctionNumber

(**************************************************************************************
 * Application   : BoxControl Framework
 * Revision date : $Date: 2013-09-23 11:26:06 +0200 (Wed, 23 Sep 2015) $
 * Author        : CDC
 * ------------------------------------------------------------------------------------
 * © Swisslog AG * Swisslog is not liable for any usage of this source code that is not agreed
 * on between Swisslog and the other party. The mandatory legal liability remains * unaffected.
 * ------------------------------------------------------------------------------------
 * Project revision history:
 *
 * VERSION DATE         INITIALS     DESCRIPTION
 * 0.0     DD.MM.YYYY   (name)       (explain customized modifications)
 *
 **************************************************************************************)

//***********************************************************************************************************
VAR_INPUT
	Name				: STRING[NAME_LENGTH]		:= '';	// name of position
END_VAR

//***********************************************************************************************************
VAR
	eFunctionNumber		: E_FunctionNumber			:= 0;
END_VAR


// string length is roughly 12chars -> hashcode is not neccessary
FOR eFunctionNumber := E_FunctionNumber.F_BEGIN_FUNCTION + 1 TO E_FunctionNumber.F_END_FUNCTION - 1 DO
	IF F_EqualSisNames(Name1:= FunctionRegistry[eFunctionNumber].FunctionName,
					 Name2:= Name) THEN
		F_FindFunction:= eFunctionNumber;
		RETURN;
	END_IF

END_FOR

// done
F_FindFunction:= E_FunctionNumber.F_BEGIN_FUNCTION;

END_FUNCTION

// ---- 20_Product/10_BCF/11_Conv/12_E_Functions/10_Helper/F_FindElement.TcPOU
// returns the element number of the element name or E_BEGIN_ELEMENT if not found
FUNCTION PUBLIC F_FindElement : E_ElementNumber

(**************************************************************************************
 * Application   : BoxControl Framework
 * Revision date : $Date: 2013-09-23 11:26:06 +0200 (Wed, 23 Sep 2015) $
 * Author        : CDC
 * ------------------------------------------------------------------------------------
 * © Swisslog AG * Swisslog is not liable for any usage of this source code that is not agreed
 * on between Swisslog and the other party. The mandatory legal liability remains * unaffected.
 * ------------------------------------------------------------------------------------
 * Project revision history:
 *
 * VERSION DATE         INITIALS     DESCRIPTION
 * 0.0     DD.MM.YYYY   (name)       (explain customized modifications)
 *
 **************************************************************************************)

//***********************************************************************************************************
VAR_INPUT
	Name				: STRING[NAME_LENGTH]		:= '';	// name of position
END_VAR

//***********************************************************************************************************
VAR
	eElementNumber		: E_ElementNumber			:= 0;
END_VAR


// string length is roughly 12chars -> hashcode is not neccessary
FOR eElementNumber := E_ElementNumber.E_BEGIN_ELEMENT + 1 TO E_ElementNumber.E_END_ELEMENT - 1 DO
	IF F_EqualSisNames(Name1:= ElementRegistry[eElementNumber].ElementName,
					 Name2:= Name) THEN
		F_FindElement:= eElementNumber;
		RETURN;
	END_IF

END_FOR

// done
F_FindElement:= E_ElementNumber.E_BEGIN_ELEMENT;

END_FUNCTION

// ---- 20_Product/10_BCF/11_Conv/12_E_Functions/10_Helper/F_FindGroup.TcPOU
// returns the group number of the group name or G_BEGIN_GROUP if not found
FUNCTION PUBLIC F_FindGroup : E_GroupNumber

(**************************************************************************************
 * Application   : BoxControl Framework
 * Revision date : $Date: 2013-09-23 11:26:06 +0200 (Wed, 23 Sep 2015) $
 * Author        : CDC
 * ------------------------------------------------------------------------------------
 * © Swisslog AG * Swisslog is not liable for any usage of this source code that is not agreed
 * on between Swisslog and the other party. The mandatory legal liability remains * unaffected.
 * ------------------------------------------------------------------------------------
 * Project revision history:
 *
 * VERSION DATE         INITIALS     DESCRIPTION
 * 0.0     DD.MM.YYYY   (name)       (explain customized modifications)
 *
 **************************************************************************************)

//***********************************************************************************************************
VAR_INPUT
  Name                  : STRING[NAME_LENGTH]         := '';    // name of position
END_VAR

//***********************************************************************************************************
VAR
  eGroupNumber          : E_GroupNumber               := 0;
END_VAR


// string length is roughly 12chars -> hashcode is not neccessary
FOR eGroupNumber := E_GroupNumber.G_BEGIN_GROUP + 1 TO E_GroupNumber.G_END_GROUP - 1 DO
	IF(F_EqualSisNames(Name1:= GroupRegistry[eGroupNumber].GroupName,
					 Name2:= Name) = TRUE)
	THEN
		F_FindGroup:= eGroupNumber;
		RETURN;
	END_IF

END_FOR

// done
F_FindGroup:= E_GroupNumber.G_BEGIN_GROUP;

END_FUNCTION

// ---- 20_Product/10_BCF/11_Conv/12_E_Functions/10_Helper/F_CheckSubsystem.TcPOU
// checks the subsystem name
FUNCTION PUBLIC F_CheckSubsystem : BOOL

(**************************************************************************************
 * Application   : BoxControl Framework
 * Revision date : $Date: 2013-09-23 11:26:06 +0200 (Wed, 23 Sep 2015) $
 * Author        : CDC
 * ------------------------------------------------------------------------------------
 * © Swisslog AG * Swisslog is not liable for any usage of this source code that is not agreed
 * on between Swisslog and the other party. The mandatory legal liability remains * unaffected.
 * ------------------------------------------------------------------------------------
 * Project revision history:
 *
 * VERSION DATE         INITIALS     DESCRIPTION
 * 0.0     DD.MM.YYYY   (name)       (explain customized modifications)
 *
 **************************************************************************************)

//***********************************************************************************************************
VAR_INPUT
  Name                  : STRING[NAME_LENGTH]         := '';    // name of position
END_VAR

//***********************************************************************************************************
VAR
END_VAR


// check name
IF F_EqualSisNames(Name1:= SubsystemRegistry.SubsystemName,
                   Name2:= Name) THEN
	F_CheckSubsystem:= TRUE;
	RETURN;
END_IF

// done
F_CheckSubsystem:= FALSE;

END_FUNCTION

// ---- 20_Product/30_Toolbox/12_StringStream/F_StuffString.TcPOU
FUNCTION F_StuffString : T_MaxString
(**************************************************************************************
 * 	Application		:	BoxControl Framework
 *	Revision		:	$Revision: 404529 $
 *	Revision date	:	$Date: 2018-04-23 08:21:38 +0200 (Mo., 23 Apr 2018) $
 *	Last changed by	:	$Author: b7bolm $
 *	URL				:	$URL: http://almscdc.swisslog.com/repo/SWPD/Development/BoxControlFramework/20_Release/trunk/01_Software/BCF/BCF/JumpStart/30_Toolbox/12_StringStream/F_StuffString.TcPOU $
 *
 *	Purpose			:	Add leading characters to get a string of predefined length.
 *						The stuffcharacter could be any character but typical '0'.
 *						The function add to the inputString acording to the input variable 
 *						Stringlenght a number of stuffCharacters.
 *
 * ------------------------------------------------------------------------------------
 *	Copyright Swisslog [IP AG], Switzerland. All rights reserved.
 * 
 * ------------------------------------------------------------------------------------
 *	
 * 	Revision History: 
 *
 * 	VERSION			DATE			INITIALS			DESCRIPTION
 *	0.1				01.01.2001		swl					Example
 *
 **************************************************************************************)
VAR_INPUT
	InputString			: STRING(MAX_STRING_LENGTH); // String to be stuffed with characters 
	StringLength		: INT; // Required string length 
	StuffCharacter		: STRING(1); // Character to stuff into string
	LeftAligned			: BOOL; // Stuff characters will be put at the end of input string
END_VAR

// Check that stuff character is valid
IF StuffCharacter <> '' THEN
	// Go through length
	WHILE LEN(InputString) < StringLength DO
		IF LeftAligned THEN
			// Fill up with trailing StuffCharacter until StringLength is reached 
			InputString := CONCAT(InputString, StuffCharacter);
		ELSE
			// Fill up with leading StuffCharacter until StringLength is reached 
			InputString := CONCAT(StuffCharacter, InputString);
		END_IF
	END_WHILE
END_IF

// Return string
F_StuffString := InputString;

END_FUNCTION

// ---- 20_Product/10_BCF/11_Conv/10_Base/F_GetTU_DataIndex.TcPOU
FUNCTION F_GetTU_DataIndex :DINT
(**************************************************************************************
 * 	Application		:	BoxControl Framework
 *	Revision		:	$Revision: 404529 $
 *	Revision date	:	$Date: 2018-04-23 08:21:38 +0200 (Mo., 23 Apr 2018) $
 *	Last changed by	:	$Author: b7bolm $
 *	URL				:	$URL: http://almscdc.swisslog.com/repo/SWPD/Development/BoxControlFramework/20_Release/trunk/01_Software/BCF/BCF/JumpStart/20_Product/10_App/10_Base/10_Lib/10_Conv/F_GetTU_DataIndex.TcPOU $
 *
 *	Purpose			:	Returns the TU - data index of a certain function.
 *
 * ------------------------------------------------------------------------------------
 *	Copyright Swisslog [IP AG], Switzerland. All rights reserved.
 * 
 * ------------------------------------------------------------------------------------
 *	
 * 	Revision History: 
 *
 * VERSION DATE         INITIALS     DESCRIPTION
 * 0.0     DD.MM.YYYY   (name)       (explain customized modifications)
 *
 **************************************************************************************)
VAR_INPUT
	eFunctionNumber		: E_FunctionNumber; // Number OF the element 
	ZoneNumber			: INT; // Zone number 
END_VAR

VAR
	DebugMsg			: T_MAXSTRING; // Debug msg
END_VAR

// Initialize
F_GetTU_DataIndex := 0;

// If a function is set 
IF eFunctionNumber > F_BEGIN_FUNCTION AND eFunctionNumber < F_END_FUNCTION
	AND ZoneNumber > 0 AND ZoneNumber <= NUMBER_OF_ZONES_PER_FUNCTION THEN
	// Check for a valid reference
	IF __ISVALIDREF(FunctionRegistry[eFunctionNumber].Zone[ZoneNumber].refZoneData) THEN
		// Return TU index
		F_GetTU_DataIndex := FunctionRegistry[eFunctionNumber].Zone[ZoneNumber].refZoneData.TransportControlData.TU_DataIndex;
	END_IF

// Invalid function index
ELSE
	//-- debug message ------------------------------------------------
	// example: '11-000-0000-00-0,  invalid function/zone number,  function = 21,  zone = 1'
	DebugMsg:= '';
	DebugMsg:= CONCAT(DebugMsg, F_AddDividerToSisString(SubsystemRegistry.SubsystemName));
	DebugMsg:= CONCAT(DebugMsg, ',  invalid function/zone number');
	DebugMsg:= CONCAT(DebugMsg, DebugTextBlocks.FUNCTIONNBR);
	DebugMsg:= CONCAT(DebugMsg, TO_STRING(eFunctionNumber));
	DebugMsg:= CONCAT(DebugMsg, DebugTextBlocks.ZONENBR);
	DebugMsg:= CONCAT(DebugMsg, INT_TO_STRING(ZoneNumber));
	fbDebugMsgManager.M_SendMessage(meMessageType:= E_DebugMsgType.ERROR,
									mDebugSource := 'F_GetTU_DataIndex', 
									mpMsgData    := ADR(DebugMsg),
									mMsgDataLen  := INT_TO_UDINT(LEN(DebugMsg)));
END_IF

END_FUNCTION

// ---- 20_Product/10_BCF/11_Conv/10_Base/F_SearchAssignmentId.TcPOU
FUNCTION F_SearchAssignmentId : DINT
(**************************************************************************************
 * 	Application		:	BoxControl Framework
 *	Revision		:	$Revision: 404529 $
 *	Revision date	:	$Date: 2018-04-23 08:21:38 +0200 (Mo., 23 Apr 2018) $
 *	Last changed by	:	$Author: b7bolm $
 *	URL				:	$URL: http://almscdc.swisslog.com/repo/SWPD/Development/BoxControlFramework/20_Release/trunk/01_Software/BCF/BCF/JumpStart/20_Product/10_App/10_Base/10_Lib/10_Conv/F_SearchAssignmentId.TcPOU $
 *
 *	Purpose			:	The function searchs searches for the AsssignementID in the TU-Data Table and then the ElementName.
 *
 * ------------------------------------------------------------------------------------
 *	Copyright Swisslog [IP AG], Switzerland. All rights reserved.
 * 
 * ------------------------------------------------------------------------------------
 *	
 * 	Revision History: 
 *
 * 	VERSION			DATE			INITIALS			DESCRIPTION
 *	0.1				01.01.2001		swl					Example
 *
 **************************************************************************************)
VAR_INPUT
	AssignmentID		: UDINT; // TU ID as string 
END_VAR

VAR
	TU_DataIndex		: DINT; // Index 
END_VAR

// Initialize
F_SearchAssignmentId := 0;

// Check assignment ID is different to UNKNOWN
IF AssignmentID = Conveyor.ASSIGNMENT_ID_UNKNOWN THEN
	// Otherwise return 0
	RETURN;
ELSIF 	AssignmentID = 0 THEN
	// Otherwise return 0
	RETURN;
END_IF

// Loop over all TU_Data sets 
FOR TU_DataIndex := 0  TO NUMBER_OF_TU_DATA DO
	// Search for equal id
	IF TU_DataTable[TU_DataIndex].AssignmentID = AssignmentID THEN
		F_SearchAssignmentId := TU_DataIndex;
		RETURN;
	END_IF
END_FOR

END_FUNCTION

// ---- 20_Product/10_BCF/11_Conv/10_Base/F_SearchTU_ByHashCode.TcPOU
// searches TU table for a specific TU and return their index if found, otherwise zero
FUNCTION PUBLIC F_SearchTU_ByHashCode : DINT

(**************************************************************************************
 * 	Application		:	BoxControl Framework
 *	Revision		:	$Revision: 404529 $
 *	Revision date	:	$Date: 2018-04-23 08:21:38 +0200 (Mo., 23 Apr 2018) $
 *	Last changed by	:	$Author: b7bolm $
 *	URL				:	$URL: http://almscdc.swisslog.com/repo/SWPD/Development/BoxControlFramework/20_Release/trunk/01_Software/BCF/BCF/JumpStart/20_Product/10_App/10_Base/10_Lib/10_Conv/F_SearchTU_ByHashCode.TcPOU $
 *
 *	Purpose			:	The function searchs searches for the TU-Data of the specified 
 *						barcode in the TU-Data Table and then the ElementName.
 *
 * ------------------------------------------------------------------------------------
 *	Copyright Swisslog [IP AG], Switzerland. All rights reserved.
 * 
 * ------------------------------------------------------------------------------------
 *	
 * 	Revision History: 
 *
 * 	VERSION			DATE			INITIALS			DESCRIPTION
 *	0.1				01.01.2001		swl					Example
 *
 **************************************************************************************)

VAR_INPUT
	TU_ID				: T_MaxString		:= '';	// TU ID as string 
END_VAR

VAR
	HashCode			: UDINT				:= 0;
	Idx					: DINT				:= 0; 
END_VAR


// valid TuID?
IF TU_ID = Conveyor.TU_ID_UNKNOWN THEN
	F_SearchTU_ByHashCode := 0;
	RETURN;
END_IF


// prepare hash code to compare
HashCode := F_CreateHashCode(TU_ID);

// Loop over all TU_Data sets 
FOR Idx := 0  TO NUMBER_OF_TU_DATA DO
	// entry used?
	IF NOT TU_DataTable[Idx].DataSet.DataPresent THEN
		CONTINUE;
	END_IF

	// hash code equal?
	IF TU_DataTable[Idx].TU_ID.HashCode <> HashCode THEN
		CONTINUE;
	END_IF

	// TU-ID equal?
	IF TU_DataTable[Idx].TU_ID.ASCII <> TU_ID THEN
		CONTINUE;
	END_IF

	// found -> return TU-Index
	F_SearchTU_ByHashCode := Idx;
	RETURN;

END_FOR

// nothing found
F_SearchTU_ByHashCode := 0;

END_FUNCTION

// ---- 20_Product/10_BCF/11_Conv/12_E_Functions/10_Helper/F_GetTransportControlData.TcPOU
FUNCTION F_GetTransportControlData : ST_TransportControlData
(**************************************************************************************
 * 	Application		:	BoxControl Framework
 *	Revision		:	$Revision: 404529 $
 *	Revision date	:	$Date: 2018-04-23 08:21:38 +0200 (Mo., 23 Apr 2018) $
 *	Last changed by	:	$Author: b7bolm $
 *	URL				:	$URL: http://almscdc.swisslog.com/repo/SWPD/Development/BoxControlFramework/20_Release/trunk/01_Software/BCF/BCF/JumpStart/20_Product/10_App/12_E_Functions/10_Lib/10_Conv/10_Functions/F_GetTransportControlData.TcPOU $
 *
 *	Purpose			:	Transport control data
 *
 * ------------------------------------------------------------------------------------
 *	Copyright Swisslog [IP AG], Switzerland. All rights reserved.
 * 
 * ------------------------------------------------------------------------------------
 *	
 * 	Revision History: 
 *
 * 	VERSION			DATE			INITIALS			DESCRIPTION
 *	0.1				01.01.2001		swl					Example
 *
 **************************************************************************************)
VAR_INPUT
	eFunctionNumber		: E_FunctionNumber; // Function number
	ZoneNumber			: INT; // Zone number
END_VAR


// Check if function number is valid
IF eFunctionNumber > E_FunctionNumber.F_BEGIN_FUNCTION AND
   eFunctionNumber < E_FunctionNumber.F_END_FUNCTION AND
   ZoneNumber > 0 THEN
  
	// Check reference is valid
	IF __ISVALIDREF(FunctionRegistry[eFunctionNumber].Zone[ZoneNumber].refZoneData) THEN
   		// Return transport control data
   		F_GetTransportControlData := FunctionRegistry[eFunctionNumber].Zone[ZoneNumber].refZoneData.TransportControlData;
	END_IF
END_IF

END_FUNCTION

// ---- 20_Product/10_BCF/11_Conv/10_Base/F_InsertTU_Data.TcPOU
FUNCTION F_InsertTU_Data : DINT
(**************************************************************************************
 * 	Application		:	BoxControl Framework
 *	Revision		:	$Revision: 404529 $
 *	Revision date	:	$Date: 2018-04-23 08:21:38 +0200 (Mo., 23 Apr 2018) $
 *	Last changed by	:	$Author: b7bolm $
 *	URL				:	$URL: http://almscdc.swisslog.com/repo/SWPD/Development/BoxControlFramework/20_Release/trunk/01_Software/BCF/BCF/JumpStart/20_Product/10_App/10_Base/10_Lib/10_Conv/F_InsertTU_Data.TcPOU $
 *
 *	Purpose			:	Searchs for a free TU-DataIndex and presets it. 
 *						Returns the TU-DataIndex. If no free TU_Data was found, it
 *						will return 0.
 *
 * ------------------------------------------------------------------------------------
 *	Copyright Swisslog [IP AG], Switzerland. All rights reserved.
 * 
 * ------------------------------------------------------------------------------------
 *	
 * 	Revision History: 
 *
 * VERSION DATE         INITIALS     DESCRIPTION
 * 0.0     DD.MM.YYYY   (name)       (explain customized modifications)
 *
 **************************************************************************************)
VAR_INPUT
	eFunctionNumber	 	: E_FunctionNumber; // Number of the function 
	ZoneNumber	 		: INT; // Number of the zone  
END_VAR

VAR
	TU_DataIndex  		: DINT; // TU-DataIndex 
	Idx	  				: INT; // Index variable 
	DebugMsg			: T_MAXSTRING; // Debug msg
	FunctionName		: STRING(NAME_LENGTH); // Function name
END_VAR

// Initialize
F_InsertTU_Data := 0;

// Search a free TU Index
FOR TU_DataIndex := 1 TO NUMBER_OF_TU_DATA BY 1 DO
	// If data set is free
	IF NOT TU_DataTable[TU_DataIndex].DataSet.DataPresent THEN
		// Return new index
		F_InsertTU_Data := TU_DataIndex;
		EXIT;
	END_IF
END_FOR

// Free index was found 
IF F_InsertTU_Data > 0 THEN
	// Set DataPresent 
	TU_DataTable[TU_DataIndex].DataSet.DataPresent := TRUE;

	// Preset TU_Data 
	TU_DataTable[TU_DataIndex].TU_ID.ASCII := Conveyor.TU_ID_UNKNOWN;
	TU_DataTable[TU_DataIndex].TU_ID.HashCode := F_CreateHashCode(Conveyor.TU_ID_UNKNOWN);
	
	// Preset Assignmetn
	TU_DataTable[TU_DataIndex].AssignmentID := Conveyor.ASSIGNMENT_ID_UNKNOWN;

	FOR Idx := 1 TO NUMBER_OF_DESTINATIONS BY 1 DO
		TU_DataTable[TU_DataIndex].Destination[Idx].eFunctionNumber := E_FunctionNumber.F_BEGIN_FUNCTION;
		TU_DataTable[TU_DataIndex].Destination[Idx].ZoneNumber := 0;
	END_FOR

	// Update time stamp 
	IF eFunctionNumber > E_FunctionNumber.F_BEGIN_FUNCTION AND
	   eFunctionNumber < E_FunctionNumber.F_END_FUNCTION THEN	
		TU_DataTable[TU_DataIndex].TimeStamp.eInsertFunctionNumber := eFunctionNumber;
	ELSE
		TU_DataTable[TU_DataIndex].TimeStamp.eInsertFunctionNumber := E_FunctionNumber.F_BEGIN_FUNCTION;
	END_IF
	
	IF ZoneNumber <= NUMBER_OF_ZONES_PER_FUNCTION THEN
		TU_DataTable[TU_DataIndex].TimeStamp.InsertZoneNumber := ZoneNumber;
	ELSE
		TU_DataTable[TU_DataIndex].TimeStamp.InsertZoneNumber := 0;	
	END_IF

	TU_DataTable[TU_DataIndex].TimeStamp.InsertDateTime := System.fbSystemTime.TIMESTR;
	
	FunctionName := F_GetFunctionName(
						eFunctionNumber := eFunctionNumber,
						ZoneNumber		:= ZoneNumber);

	//-- debug message ------------------------------------------------
	// example: '11-001-1979-01-9,  TU_Data inserted,  TU_DataIndex = 1979,  TuID = 0012345600,  AssignmentID = 19790109'
	DebugMsg:= '';
	DebugMsg:= CONCAT(DebugMsg, F_AddDividerToSisString(FunctionName));
	DebugMsg:= CONCAT(DebugMsg, ',  TU_Data inserted');
	DebugMsg:= CONCAT(DebugMsg, F_CreateTU_DataString(TU_DataIndex));
	fbDebugMsgManager.M_SendMessage(meMessageType:= E_DebugMsgType.INFO,
									mDebugSource := 'F_InsertTU_Data', 
									mpMsgData    := ADR(DebugMsg),
									mMsgDataLen  := INT_TO_UDINT(LEN(DebugMsg)));
END_IF

END_FUNCTION

